// TIA Portal V20 export
FUNCTION_BLOCK "CallEquipment"   // FB43, LAD
TITLE = CallEquipment
// This block includes all general functions, checks and logik that is needed in the entire unit. E.g. general releases and system wide functionalities like air, pressure and power handling as well as general reaction to events.
// stored: IsIECCheckEnabled true, MemoryReserve 100, Namespace Unit1.Em5, SetENOAutomatically true
   VAR_INPUT
      ZoneOperationEnable { ExternalWritable := 'False'} : "LWONIK_typeSafetyZoneManualOperation";
   END_VAR
   VAR_IN_OUT
      unitStatus : "LAF_typeUnitStatus";   // Current unit status o be used in this EM
      emFeedback : "LUC_typeEmFeedback";   // Feedback of the EM to the Unit
      unitAlarmDB : "LAF_typeAlarms";   // Summarized EM Alarms for the Unit
   END_VAR
   VAR
      InstSequenceTransferPnPLeft { ExternalWritable := 'False'} : "Unit1.Em5.Sequence_1_TransferPnPLeft";
      InstSequenceTransferPnPRight { ExternalWritable := 'False'} : "Unit1.Em5.Sequence_2_TransferPnPRight";
      InstSequenceGaugeRnR { ExternalWritable := 'False'} : "Unit1.Em5.Sequence_10_GaugeRnR";
      instTransferPnPLeftHomeJob1 { ExternalWritable := 'False'} : "LAF_SelectJob";
      instTransferPnPLeftSideTapeLoadJob2 { ExternalWritable := 'False'} : "LAF_SelectJob";
      instTransferPnPLeftHotPressLeftUnloadJob3 { ExternalWritable := 'False'} : "LAF_SelectJob";
      instTransferPnPLeftHotPressLeftLoadJob4 { ExternalWritable := 'False'} : "LAF_SelectJob";
      instTransferPnPLeftSideTapeLoadJob5 { ExternalWritable := 'False'} : "LAF_SelectJob";
      instTransferPnPLeftHotPressRightUnloadJob6 { ExternalWritable := 'False'} : "LAF_SelectJob";
      instTransferPnPLeftHotPressRightLoadJob7 { ExternalWritable := 'False'} : "LAF_SelectJob";
      instTransferPnPLeftHipotThicknessUnloadJob9 { ExternalWritable := 'False'} : "LAF_SelectJob";
      instTransferPnPRightHomeJob1 { ExternalWritable := 'False'} : "LAF_SelectJob";
      instTransferPnPRightHipotThicknessLoadJob2 { ExternalWritable := 'False'} : "LAF_SelectJob";
      instTransferPnPRightVisionUnloadJob3 { ExternalWritable := 'False'} : "LAF_SelectJob";
      instTransferPnPRightVisionLoadJob4 { ExternalWritable := 'False'} : "LAF_SelectJob";
      instTransferPnPRightLaserMarkUnloadJob5 { ExternalWritable := 'False'} : "LAF_SelectJob";
      instTransferPnPRightLaserMarkLoadJob6 { ExternalWritable := 'False'} : "LAF_SelectJob";
      instTransferPnPRightWeightCheckUnloadJob9 { ExternalWritable := 'False'} : "LAF_SelectJob";
      instGRnR_SideTapeLoadJob2_Left { ExternalWritable := 'False'} : "LAF_SelectJob";
      instGRnR_HipotThicknessUnloadJob3_Left { ExternalWritable := 'False'} : "LAF_SelectJob";
      instGRnR_HipotThicknessLoadJob4_Left { ExternalWritable := 'False'} : "LAF_SelectJob";
      instGRnR_HipotThicknessLoadJob5_Right { ExternalWritable := 'False'} : "LAF_SelectJob";
      instGRnR_VisionUnloadJob6_Right { ExternalWritable := 'False'} : "LAF_SelectJob";
      instGRnR_VisionLoadJob7_Right { ExternalWritable := 'False'} : "LAF_SelectJob";
      instGRnR_WeightCheckUnloadJob8_Right { ExternalWritable := 'False'} : "LAF_SelectJob";
      instGRnR_WeightCheckLoadJob9_Right { ExternalWritable := 'False'} : "LAF_SelectJob";
      instCmTransferPnPLeftSafetyPin { ExternalWritable := 'False'} : "LBC_DigitalSignalCn";
      instCmTransferPnPLeftJRDetect { ExternalWritable := 'False'} : "LBC_DigitalSignalCn";
      instCmTransferPnPRightSafetyPin { ExternalWritable := 'False'} : "LBC_DigitalSignalCn";
      instCmTransferPnPRightJRDetect { ExternalWritable := 'False'} : "LBC_DigitalSignalCn";
      instCmTransferPnPLeftAxisX { ExternalWritable := 'False'} : "LBC_Axis64Pos_TecPlcCn";
      instCmTransferPnPLeftAxisY { ExternalWritable := 'False'} : "LBC_Axis64Pos_TecPlcCn";
      instCmTransferPnPLeftAxisZ { ExternalWritable := 'False'} : "LBC_Axis64Pos_TecPlcCn";
      instCmTransferPnPRightAxisX { ExternalWritable := 'False'} : "LBC_Axis64Pos_TecPlcCn";
      instCmTransferPnPRightAxisY { ExternalWritable := 'False'} : "LBC_Axis64Pos_TecPlcCn";
      instCmTransferPnPRightAxisZ { ExternalWritable := 'False'} : "LBC_Axis64Pos_TecPlcCn";
      instCmTransferPnPLeftClampOpenClose { ExternalWritable := 'False'} : "LBC_TwoWayActuatorCn";
      instCmTransferPnPRightClampOpenClose { ExternalWritable := 'False'} : "LBC_TwoWayActuatorCn";
      instInterlockTransferPnPLeftAxisX { ExternalWritable := 'False'} : "LER_Axis64Pos_InterlockSummary";
      instInterlockTransferPnPLeftAxisY { ExternalWritable := 'False'} : "LER_Axis64Pos_InterlockSummary";
      instInterlockTransferPnPLeftAxisZ { ExternalWritable := 'False'} : "LER_Axis64Pos_InterlockSummary";
      instInterlockTransferPnPRightAxisX { ExternalWritable := 'False'} : "LER_Axis64Pos_InterlockSummary";
      instInterlockTransferPnPRightAxisY { ExternalWritable := 'False'} : "LER_Axis64Pos_InterlockSummary";
      instInterlockTransferPnPRightAxisZ { ExternalWritable := 'False'} : "LER_Axis64Pos_InterlockSummary";
      instLDrv701ControlTransferPnPLeftAxisZ { ExternalWritable := 'False'} : "LDrvSafe_SinaTlg701Control";   // Drive Telegram Function Library
      instLDrv701StatusTransferPnPLeftAxisZ { ExternalWritable := 'False'} : "LDrvSafe_SinaTlg701Status";   // Drive Telegram Function Library
      instLDrv701ControlTransferPnPRightAxisZ { ExternalWritable := 'False'} : "LDrvSafe_SinaTlg701Control";   // Drive Telegram Function Library
      instLDrv701StatusTransferPnPRightAxisZ { ExternalWritable := 'False'} : "LDrvSafe_SinaTlg701Status";   // Drive Telegram Function Library
      instManageAlarms { ExternalWritable := 'False'} : "LAF_ManageAlarms";
      instEventsPFE { ExternalWritable := 'False'} : "Unit1.Em5.EventsPFE";
      statUnitStatus { ExternalWritable := 'False'} : "LAF_typeUnitStatus";   // Unit Status that is used in this project
      statSlmStatus { ExternalWritable := 'False'} : Struct
         running : Bool;
         powerOff : Bool;
      END_STRUCT;
      statAllBrakeTest { ExternalWritable := 'False'} : "LER_typeBrakeTestUnitCommands";
      statFlipFlop { ExternalWritable := 'False'} : Array[0..99] of Bool;
      statPartData { ExternalWritable := 'False'} : "LER_typePartData";
      statDataDelete { ExternalWritable := 'False'} : "LER_typePartData";
      statRoutingOk { ExternalWritable := 'False'} : Array[0..99] of Bool;
      statRoutingNok { ExternalWritable := 'False'} : Array[0..99] of Bool;
      statTonTime { ExternalWritable := 'False'} : Array[0..999] of TON_TIME;
      statTofTime { ExternalWritable := 'False'} : Array[0..99] of TOF_TIME;
      statPulse { ExternalWritable := 'False'} : Array[0..999] of Bool;
      statTrPnP_GaugeRnR : Struct
         currentCount : Int;
         processCount : Int;
         Ongoing : Bool;
         Complete : Bool;
      END_STRUCT;
      statEnableManualCmds { ExternalWritable := 'False'} : Bool;
      "*** Interlock Axis ***" : Bool;
      TransferPnPLeftAxisX_Home { S7_SetPoint := 'True'} : "LER_Axis_Homing";
      TransferPnPLeftAxisY_Home { S7_SetPoint := 'True'} : "LER_Axis_Homing";
      TransferPnPLeftAxisZ_Home { S7_SetPoint := 'True'} : "LER_Axis_Homing";
      TransferPnPRightAxisX_Home { S7_SetPoint := 'True'} : "LER_Axis_Homing";
      TransferPnPRightAxisY_Home { S7_SetPoint := 'True'} : "LER_Axis_Homing";
      TransferPnPRightAxisZ_Home { S7_SetPoint := 'True'} : "LER_Axis_Homing";
      TransferPnPLeftAxisX_IntHome : Array[0..9] of Bool;
      TransferPnPLeftAxisY_IntHome : Array[0..9] of Bool;
      TransferPnPLeftAxisZ_IntHome : Array[0..9] of Bool;
      TransferPnPRightAxisX_IntHome : Array[0..9] of Bool;
      TransferPnPRightAxisY_IntHome : Array[0..9] of Bool;
      TransferPnPRightAxisZ_IntHome : Array[0..9] of Bool;
      TransferPnPLeftAxisX_Jog { S7_SetPoint := 'True'} : Array[0..2] of "LER_Axis_Jog";
      TransferPnPLeftAxisY_Jog { S7_SetPoint := 'True'} : Array[0..2] of "LER_Axis_Jog";
      TransferPnPLeftAxisZ_Jog { S7_SetPoint := 'True'} : Array[0..2] of "LER_Axis_Jog";
      TransferPnPRightAxisX_Jog { S7_SetPoint := 'True'} : Array[0..2] of "LER_Axis_Jog";
      TransferPnPRightAxisY_Jog { S7_SetPoint := 'True'} : Array[0..2] of "LER_Axis_Jog";
      TransferPnPRightAxisZ_Jog { S7_SetPoint := 'True'} : Array[0..2] of "LER_Axis_Jog";
      TransferPnPLeftAxisX_interlock { S7_SetPoint := 'True'} : Array[0..10] of "LER_Axis_Absolute";
      TransferPnPLeftAxisY_interlock { S7_SetPoint := 'True'} : Array[0..10] of "LER_Axis_Absolute";
      TransferPnPLeftAxisZ_interlock { S7_SetPoint := 'True'} : Array[0..10] of "LER_Axis_Absolute";
      TransferPnPRightAxisX_interlock { S7_SetPoint := 'True'} : Array[0..10] of "LER_Axis_Absolute";
      TransferPnPRightAxisY_interlock { S7_SetPoint := 'True'} : Array[0..10] of "LER_Axis_Absolute";
      TransferPnPRightAxisZ_interlock { S7_SetPoint := 'True'} : Array[0..10] of "LER_Axis_Absolute";
      TransferPnPLeftAxisX_IntPos : Array[0..9] of Struct
         "Int" : Array[1..10] of Bool;
      END_STRUCT;
      TransferPnPLeftAxisY_IntPos : Array[0..9] of Struct
         "Int" : Array[1..10] of Bool;
      END_STRUCT;
      TransferPnPLeftAxisZ_IntPos : Array[0..9] of Struct
         "Int" : Array[1..10] of Bool;
      END_STRUCT;
      TransferPnPRightAxisX_IntPos : Array[0..9] of Struct
         "Int" : Array[1..10] of Bool;
      END_STRUCT;
      TransferPnPRightAxisY_IntPos : Array[0..9] of Struct
         "Int" : Array[1..10] of Bool;
      END_STRUCT;
      TransferPnPRightAxisZ_IntPos : Array[0..9] of Struct
         "Int" : Array[1..10] of Bool;
      END_STRUCT;
      "*** Interlock TwoWay ***" { S7_SetPoint := 'True'} : "LER_Axis_Homing";
      instCmTransferPnPLeftClampOpenCloseInterlock { S7_SetPoint := 'True'} : Array[0..2] of "LER_Actuator";
      instCmTransferPnPRightClampOpenCloseInterlock { S7_SetPoint := 'True'} : Array[0..2] of "LER_Actuator";
      TransferPnPLeftClampOpenClose_Inpos : Array[0..2] of Struct
         "Int" : Array[1..10] of Bool;
      END_STRUCT;
      TransferPnPRightClampOpenClose_Inpos : Array[0..2] of Struct
         "Int" : Array[1..10] of Bool;
      END_STRUCT;
      citi_Ptrig : Array[0..20] of Bool;
      citiTon : Array[0..20] of TON_TIME;
      citi : Time;
      citiTest : Array[0..20] of Bool;
   END_VAR
   VAR_TEMP
      tempScInProduction : Bool;   // Mode Production and StateComplete
      tempScNoProduction : Bool;   // Mode Manual and StateComplete
      tempPnPLeftPart_No_Detect : Bool;
      tempPnPRightPart_No_Detect : Bool;
      tempPnPLeftPart_Detect : Bool;
      tempPnPRightPart_Detect : Bool;
      tempGuageRnR_1CycleDone : Bool;
      tempSpecialFunctionCheckbit : Bool;
      tempInterlockCond : Bool;
      tempPickCond : Bool;
      tempPlaceCond : Bool;
   END_VAR
   VAR CONSTANT
      delayTime : Time := T#3s;
      TRUE : Bool := TRUE;
      FALSE : Bool := FALSE;
      NO_JOB : DInt;
      MIN_POSITION_NUMBER : SInt;
      INIT_POSITION_NUMBER : SInt := -1;
      Stacker1 : Char := 'A';
      Stacker2 : Char := 'B';
   END_VAR
   VAR_TEMP   // added for the SCL form of the ladder/FBD networks
      _w1 : Bool;
      _w2 : Bool;
      _w3 : Bool;
      _w4 : Bool;
      _w5 : Bool;
      _w6 : Bool;
      _w7 : Bool;
      _w8 : Bool;
      _w9 : Bool;
      _w10 : Bool;
      _w11 : Bool;
      _w12 : Bool;
      _w13 : Bool;
      _w14 : Bool;
      _w15 : Bool;
      _w16 : Bool;
   END_VAR
BEGIN

REGION Network 1: BLOCK INFO HEADER
   // (company) / (C) Copyright (year)
   // ---------------------------------------------------------------------------------
   // Title:                             (Title of this block)
   // Comment/Function: (that is implemented in the block)
   // Library/Family:           (that the source is dedicated to)
   // Author:                        (department / person in charge / contact)
   // Target System:          (test system with FW version)
   // Engineering:              TIA Portal (SW version)
   // Restrictions:               (OB types, etc.)
   // Requirements:           (hardware, technological package, etc.)
   // ---------------------------------------------------------------------------------
   // Change log table:
   // Version          | Date             | Signature      | Expert in charge  | Changes applied ------------------------|----------------------|-------------------------|--------------------------------|-----------------------
   // 001.000.000 | yyyy-mm-dd | 0x00000000 | (name of expert) | First released version
END_REGION

REGION Network 2: DESCRIPTION
   // This is a template block provided by the Automation Framework. It can be used to create an own project.
   // The Block Info Header is prepared to put in your own data.
   // Description of the block could be added here and the docu created by Code2Docu.
END_REGION

REGION Network 3: Simulation
   // If simulation is active on a global level, inherit this status and set simulation active in this unit also. Information is written to DB ControlNodes, from where it is distributed to the equipmemt modules.
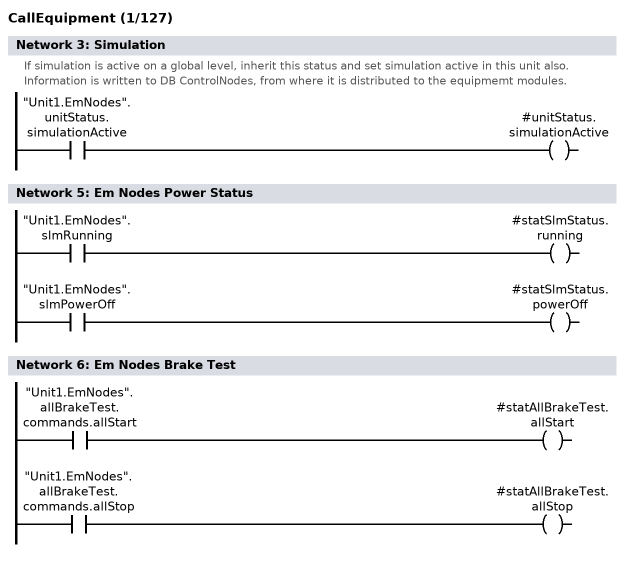
   RUNG wire#powerrail
      Contact( "Unit1.EmNodes".unitStatus.simulationActive )
      Coil( #unitStatus.simulationActive )
   END_RUNG
   // the same network as SCL:
   #unitStatus.simulationActive := "Unit1.EmNodes".unitStatus.simulationActive;
END_REGION

REGION Network 4: ******************** Unit Input ********************
END_REGION

REGION Network 5: Em Nodes Power Status
   RUNG wire#powerrail
      Contact( "Unit1.EmNodes".slmRunning )
      Coil( #statSlmStatus.running )
   END_RUNG
   RUNG wire#powerrail
      Contact( "Unit1.EmNodes".slmPowerOff )
      Coil( #statSlmStatus.powerOff )
   END_RUNG
   // the same network as SCL:
   #statSlmStatus.running := "Unit1.EmNodes".slmRunning;
   #statSlmStatus.powerOff := "Unit1.EmNodes".slmPowerOff;
END_REGION

REGION Network 6: Em Nodes Brake Test
   RUNG wire#powerrail
      Contact( "Unit1.EmNodes".allBrakeTest.commands.allStart )
      Coil( #statAllBrakeTest.allStart )
   END_RUNG
   RUNG wire#powerrail
      Contact( "Unit1.EmNodes".allBrakeTest.commands.allStop )
      Coil( #statAllBrakeTest.allStop )
   END_RUNG
   // the same network as SCL:
   #statAllBrakeTest.allStart := "Unit1.EmNodes".allBrakeTest.commands.allStart;
   #statAllBrakeTest.allStop := "Unit1.EmNodes".allBrakeTest.commands.allStop;
END_REGION

REGION Network 7: Em Data
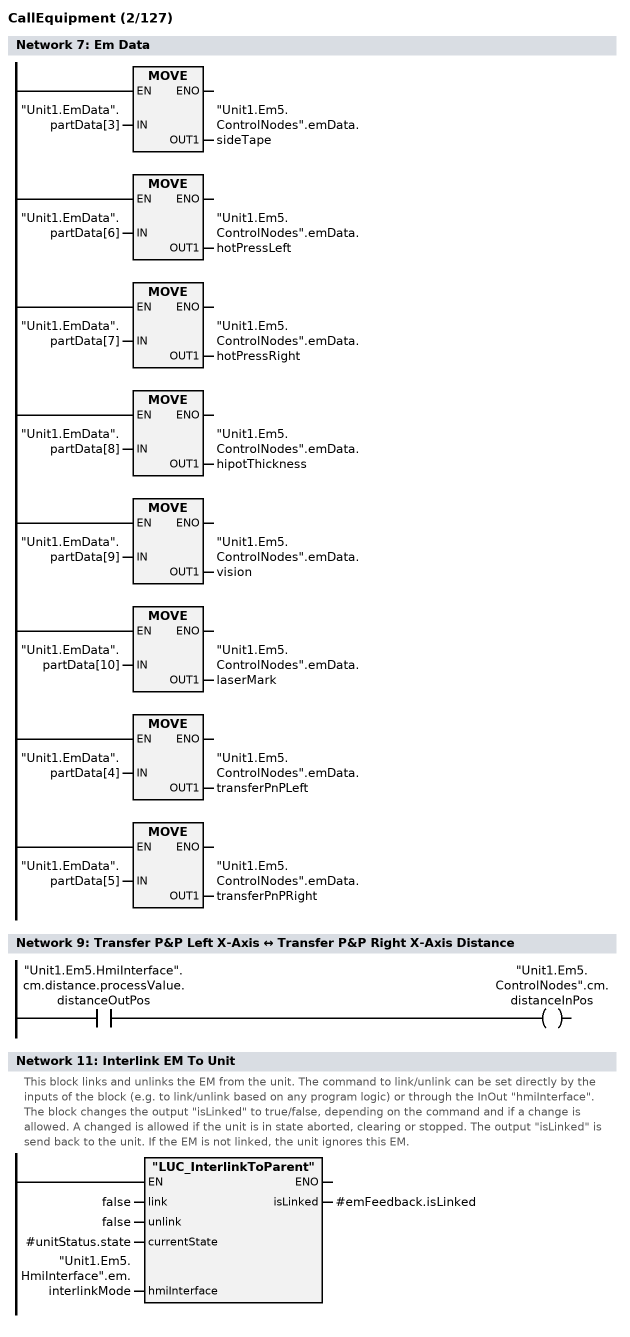
   RUNG wire#powerrail
      Move(in := "Unit1.EmData".partData[3], out1 => "Unit1.Em5.ControlNodes".emData.sideTape)
   END_RUNG
   RUNG wire#powerrail
      Move(in := "Unit1.EmData".partData[6], out1 => "Unit1.Em5.ControlNodes".emData.hotPressLeft)
   END_RUNG
   RUNG wire#powerrail
      Move(in := "Unit1.EmData".partData[7], out1 => "Unit1.Em5.ControlNodes".emData.hotPressRight)
   END_RUNG
   RUNG wire#powerrail
      Move(in := "Unit1.EmData".partData[8], out1 => "Unit1.Em5.ControlNodes".emData.hipotThickness)
   END_RUNG
   RUNG wire#powerrail
      Move(in := "Unit1.EmData".partData[9], out1 => "Unit1.Em5.ControlNodes".emData.vision)
   END_RUNG
   RUNG wire#powerrail
      Move(in := "Unit1.EmData".partData[10], out1 => "Unit1.Em5.ControlNodes".emData.laserMark)
   END_RUNG
   RUNG wire#powerrail
      Move(in := "Unit1.EmData".partData[4], out1 => "Unit1.Em5.ControlNodes".emData.transferPnPLeft)
   END_RUNG
   RUNG wire#powerrail
      Move(in := "Unit1.EmData".partData[5], out1 => "Unit1.Em5.ControlNodes".emData.transferPnPRight)
   END_RUNG
   // the same network as SCL:
   "Unit1.Em5.ControlNodes".emData.sideTape := "Unit1.EmData".partData[3];
   "Unit1.Em5.ControlNodes".emData.hotPressLeft := "Unit1.EmData".partData[6];
   "Unit1.Em5.ControlNodes".emData.hotPressRight := "Unit1.EmData".partData[7];
   "Unit1.Em5.ControlNodes".emData.hipotThickness := "Unit1.EmData".partData[8];
   "Unit1.Em5.ControlNodes".emData.vision := "Unit1.EmData".partData[9];
   "Unit1.Em5.ControlNodes".emData.laserMark := "Unit1.EmData".partData[10];
   "Unit1.Em5.ControlNodes".emData.transferPnPLeft := "Unit1.EmData".partData[4];
   "Unit1.Em5.ControlNodes".emData.transferPnPRight := "Unit1.EmData".partData[5];
END_REGION

REGION Network 8: ******************** HmiInterface → ControlNode ********************
END_REGION

REGION Network 9: Transfer P&P Left X-Axis ↔ Transfer P&P Right X-Axis Distance
   RUNG wire#powerrail
      Contact( "Unit1.Em5.HmiInterface".cm.distance.processValue.distanceOutPos )
      Coil( "Unit1.Em5.ControlNodes".cm.distanceInPos )
   END_RUNG
   // the same network as SCL:
   "Unit1.Em5.ControlNodes".cm.distanceInPos := "Unit1.Em5.HmiInterface".cm.distance.processValue.distanceOutPos;
END_REGION

REGION Network 10: ******************** Equipment Control ********************
END_REGION

REGION Network 11: Interlink EM To Unit
   // This block links and unlinks the EM from the unit. The command to link/unlink can be set directly by the inputs of the block (e.g. to link/unlink based on any program logic) or through the InOut "hmiInterface". The block changes the output "isLinked" to true/false, depending on the command and if a change is allowed. A changed is allowed if the unit is in state aborted, clearing or stopped. The output "isLinked" is send back to the unit. If the EM is not linked, the unit ignores this EM.
   RUNG wire#powerrail
      "LUC_InterlinkToParent"(link := false, unlink := false, currentState := #unitStatus.state, hmiInterface := "Unit1.Em5.HmiInterface".em.interlinkMode, isLinked => #emFeedback.isLinked)
   END_RUNG
   // the same network as SCL:
   "LUC_InterlinkToParent"(link := false,
                           unlink := false,
                           currentState := #unitStatus.state,
                           hmiInterface := "Unit1.Em5.HmiInterface".em.interlinkMode,
                           isLinked => #emFeedback.isLinked);
END_REGION

REGION Network 12: Control EM
   // When linked, unitStatus is fully applied to unitStatusUsed.
   // When not linked, only acknowledge and safetyReleased from the unitStatus are applied. A direct EM control by hmiInterface or localInterface is possible.
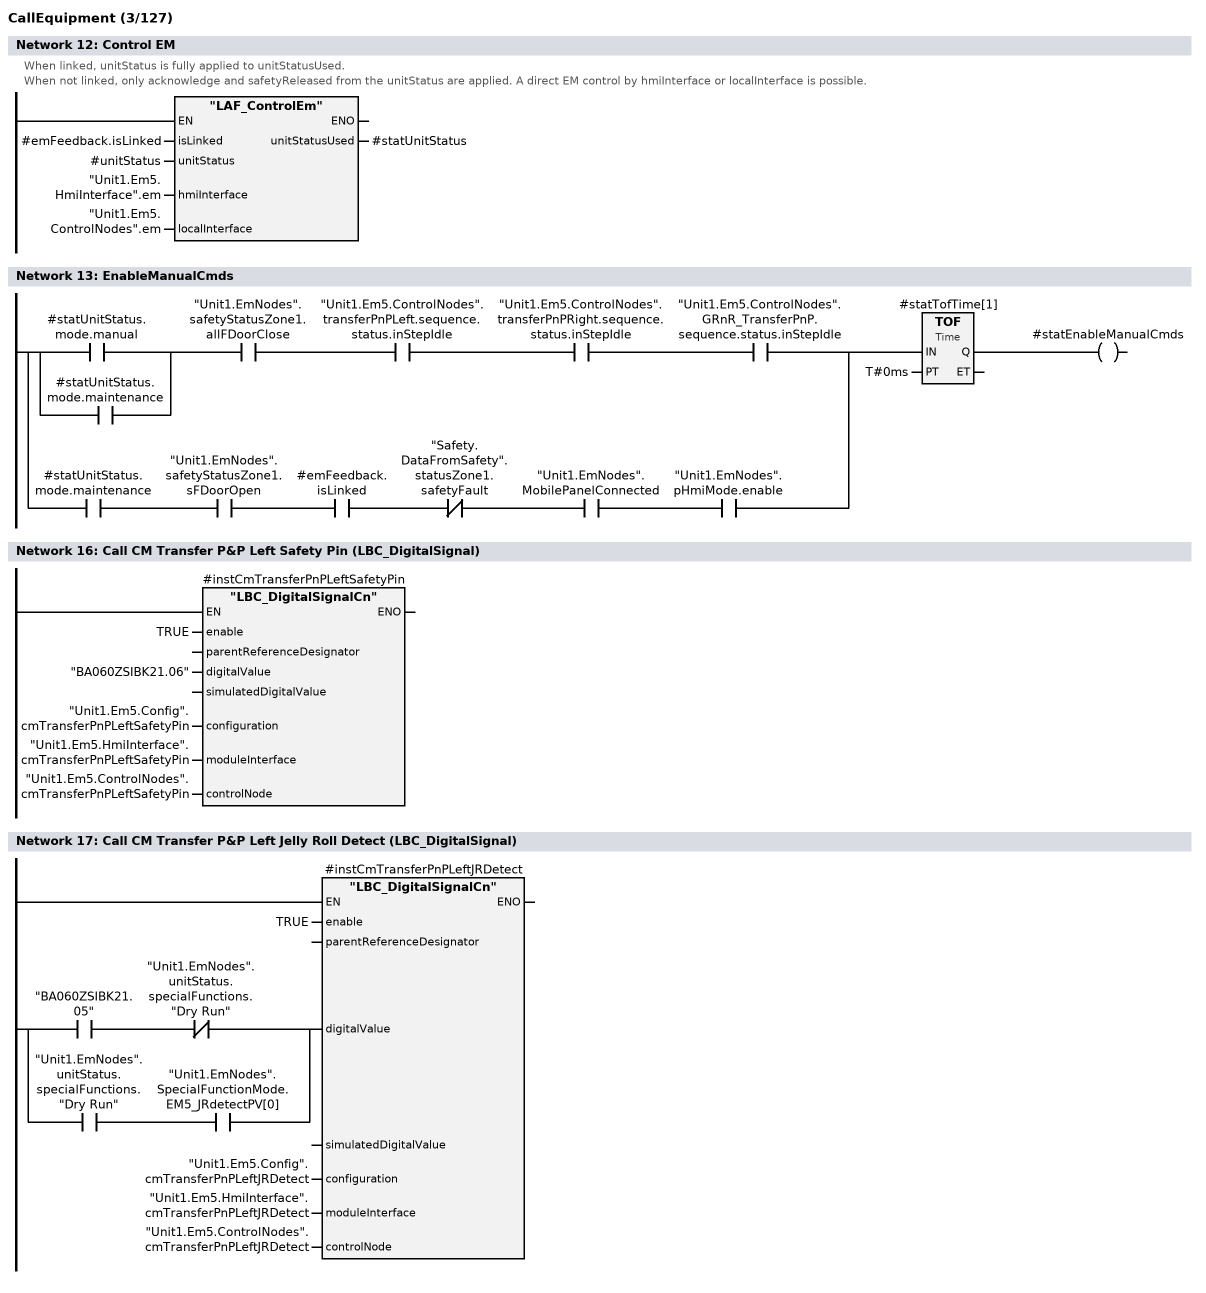
   RUNG wire#powerrail
      "LAF_ControlEm"(isLinked := #emFeedback.isLinked, unitStatus := #unitStatus, hmiInterface := "Unit1.Em5.HmiInterface".em, localInterface := "Unit1.Em5.ControlNodes".em, unitStatusUsed => #statUnitStatus)
   END_RUNG
   // the same network as SCL:
   "LAF_ControlEm"(isLinked := #emFeedback.isLinked,
                   unitStatus := #unitStatus,
                   hmiInterface := "Unit1.Em5.HmiInterface".em,
                   localInterface := "Unit1.Em5.ControlNodes".em,
                   unitStatusUsed => #statUnitStatus);
END_REGION

REGION Network 13: EnableManualCmds
   RUNG wire#powerrail
      Contact( #statUnitStatus.mode.manual )
      wire#w1
      Contact( "Unit1.EmNodes".safetyStatusZone1.allFDoorClose )
      Contact( "Unit1.Em5.ControlNodes".transferPnPLeft.sequence.status.inStepIdle )
      Contact( "Unit1.Em5.ControlNodes".transferPnPRight.sequence.status.inStepIdle )
      Contact( "Unit1.Em5.ControlNodes".GRnR_TransferPnP.sequence.status.inStepIdle )
      wire#w2
      { S7_Templates := "time_type := Time" } #statTofTime[1].TOF(pt := T#0ms, et =>)
      Coil( #statEnableManualCmds )
   END_RUNG
   RUNG wire#powerrail
      Contact( #statUnitStatus.mode.maintenance )
   END_RUNG wire#w1
   RUNG wire#powerrail
      Contact( #statUnitStatus.mode.maintenance )
      Contact( "Unit1.EmNodes".safetyStatusZone1.sFDoorOpen )
      Contact( #emFeedback.isLinked )
      I_Contact( "Safety.DataFromSafety".statusZone1.safetyFault )
      Contact( "Unit1.EmNodes".MobilePanelConnected )
      Contact( "Unit1.EmNodes".pHmiMode.enable )
   END_RUNG wire#w2
   // the same network as SCL:
   #statTofTime[1].TOF(IN := ((#statUnitStatus.mode.manual OR #statUnitStatus.mode.maintenance) AND "Unit1.EmNodes".safetyStatusZone1.allFDoorClose AND "Unit1.Em5.ControlNodes".transferPnPLeft.sequence.status.inStepIdle AND "Unit1.Em5.ControlNodes".transferPnPRight.sequence.status.inStepIdle AND "Unit1.Em5.ControlNodes".GRnR_TransferPnP.sequence.status.inStepIdle) OR (#statUnitStatus.mode.maintenance AND "Unit1.EmNodes".safetyStatusZone1.sFDoorOpen AND #emFeedback.isLinked AND NOT "Safety.DataFromSafety".statusZone1.safetyFault AND "Unit1.EmNodes".MobilePanelConnected AND "Unit1.EmNodes".pHmiMode.enable),
                       PT := T#0ms);
   #statEnableManualCmds := #statTofTime[1].Q;
END_REGION

REGION Network 15: ******************** Control Modules (Sensors) ********************
   // Call control modules that are sensors before the em logic (jobs and sequence), so that the latest value is used in the logic.
END_REGION

REGION Network 16: Call CM Transfer P&P Left Safety Pin (LBC_DigitalSignal)
   RUNG wire#powerrail
      #instCmTransferPnPLeftSafetyPin(enable := TRUE, parentReferenceDesignator :=, digitalValue := "BA060ZSIBK21.06", simulatedDigitalValue :=, configuration := "Unit1.Em5.Config".cmTransferPnPLeftSafetyPin, moduleInterface := "Unit1.Em5.HmiInterface".cmTransferPnPLeftSafetyPin, controlNode := "Unit1.Em5.ControlNodes".cmTransferPnPLeftSafetyPin)
   END_RUNG
   // the same network as SCL:
   #instCmTransferPnPLeftSafetyPin(enable := TRUE,   // "LBC_DigitalSignalCn"
                           digitalValue := "BA060ZSIBK21.06",
                           configuration := "Unit1.Em5.Config".cmTransferPnPLeftSafetyPin,
                           moduleInterface := "Unit1.Em5.HmiInterface".cmTransferPnPLeftSafetyPin,
                           controlNode := "Unit1.Em5.ControlNodes".cmTransferPnPLeftSafetyPin);
END_REGION

REGION Network 17: Call CM Transfer P&P Left Jelly Roll Detect (LBC_DigitalSignal)
   RUNG wire#powerrail
      #instCmTransferPnPLeftJRDetect(digitalValue := wire#w1, enable := TRUE, parentReferenceDesignator :=, simulatedDigitalValue :=, configuration := "Unit1.Em5.Config".cmTransferPnPLeftJRDetect, moduleInterface := "Unit1.Em5.HmiInterface".cmTransferPnPLeftJRDetect, controlNode := "Unit1.Em5.ControlNodes".cmTransferPnPLeftJRDetect)
   END_RUNG
   RUNG wire#powerrail
      Contact( "BA060ZSIBK21.05" )
      I_Contact( "Unit1.EmNodes".unitStatus.specialFunctions."Dry Run" )
   END_RUNG wire#w1
   RUNG wire#powerrail
      Contact( "Unit1.EmNodes".unitStatus.specialFunctions."Dry Run" )
      Contact( "Unit1.EmNodes".SpecialFunctionMode.EM5_JRdetectPV[0] )
   END_RUNG wire#w1
   // the same network as SCL:
   #instCmTransferPnPLeftJRDetect(enable := TRUE,   // "LBC_DigitalSignalCn"
                           digitalValue := ("BA060ZSIBK21.05" AND NOT "Unit1.EmNodes".unitStatus.specialFunctions."Dry Run") OR ("Unit1.EmNodes".unitStatus.specialFunctions."Dry Run" AND "Unit1.EmNodes".SpecialFunctionMode.EM5_JRdetectPV[0]),
                           configuration := "Unit1.Em5.Config".cmTransferPnPLeftJRDetect,
                           moduleInterface := "Unit1.Em5.HmiInterface".cmTransferPnPLeftJRDetect,
                           controlNode := "Unit1.Em5.ControlNodes".cmTransferPnPLeftJRDetect);
END_REGION

REGION Network 18: Call CM Transfer P&P Right Safety Pin (LBC_DigitalSignal)
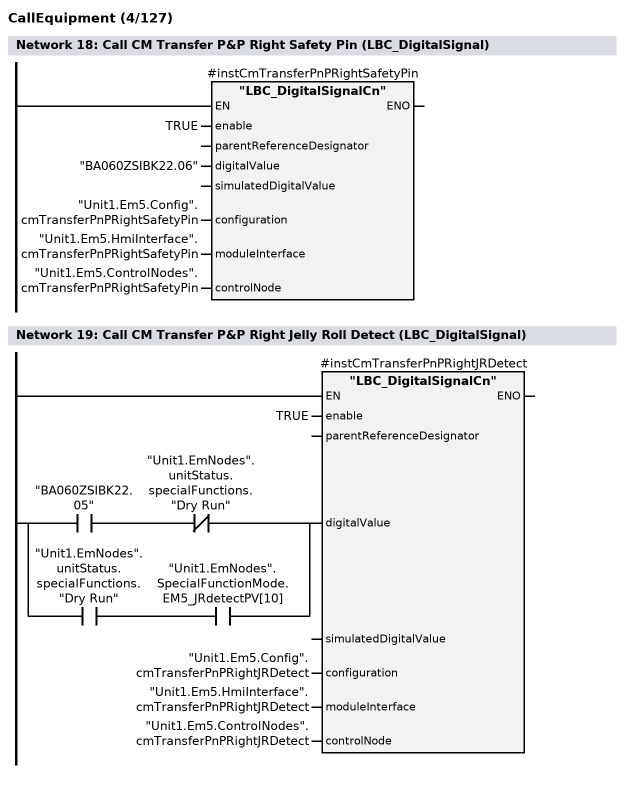
   RUNG wire#powerrail
      #instCmTransferPnPRightSafetyPin(enable := TRUE, parentReferenceDesignator :=, digitalValue := "BA060ZSIBK22.06", simulatedDigitalValue :=, configuration := "Unit1.Em5.Config".cmTransferPnPRightSafetyPin, moduleInterface := "Unit1.Em5.HmiInterface".cmTransferPnPRightSafetyPin, controlNode := "Unit1.Em5.ControlNodes".cmTransferPnPRightSafetyPin)
   END_RUNG
   // the same network as SCL:
   #instCmTransferPnPRightSafetyPin(enable := TRUE,   // "LBC_DigitalSignalCn"
                           digitalValue := "BA060ZSIBK22.06",
                           configuration := "Unit1.Em5.Config".cmTransferPnPRightSafetyPin,
                           moduleInterface := "Unit1.Em5.HmiInterface".cmTransferPnPRightSafetyPin,
                           controlNode := "Unit1.Em5.ControlNodes".cmTransferPnPRightSafetyPin);
END_REGION

REGION Network 19: Call CM Transfer P&P Right Jelly Roll Detect (LBC_DigitalSignal)
   RUNG wire#powerrail
      #instCmTransferPnPRightJRDetect(digitalValue := wire#w1, enable := TRUE, parentReferenceDesignator :=, simulatedDigitalValue :=, configuration := "Unit1.Em5.Config".cmTransferPnPRightJRDetect, moduleInterface := "Unit1.Em5.HmiInterface".cmTransferPnPRightJRDetect, controlNode := "Unit1.Em5.ControlNodes".cmTransferPnPRightJRDetect)
   END_RUNG
   RUNG wire#powerrail
      Contact( "BA060ZSIBK22.05" )
      I_Contact( "Unit1.EmNodes".unitStatus.specialFunctions."Dry Run" )
   END_RUNG wire#w1
   RUNG wire#powerrail
      Contact( "Unit1.EmNodes".unitStatus.specialFunctions."Dry Run" )
      Contact( "Unit1.EmNodes".SpecialFunctionMode.EM5_JRdetectPV[10] )
   END_RUNG wire#w1
   // the same network as SCL:
   #instCmTransferPnPRightJRDetect(enable := TRUE,   // "LBC_DigitalSignalCn"
                           digitalValue := ("BA060ZSIBK22.05" AND NOT "Unit1.EmNodes".unitStatus.specialFunctions."Dry Run") OR ("Unit1.EmNodes".unitStatus.specialFunctions."Dry Run" AND "Unit1.EmNodes".SpecialFunctionMode.EM5_JRdetectPV[10]),
                           configuration := "Unit1.Em5.Config".cmTransferPnPRightJRDetect,
                           moduleInterface := "Unit1.Em5.HmiInterface".cmTransferPnPRightJRDetect,
                           controlNode := "Unit1.Em5.ControlNodes".cmTransferPnPRightJRDetect);
END_REGION

REGION Network 21: ******************** Equipment seuqnece logic ********************
END_REGION

REGION Network 22: Map Unit Status To Sequence Status
   // This block maps the unit status to the seuqnce status. Thus, it controls the sequence depending on the unit status. E.g. it sets the sequence to automatic when the unit state is in productions. This blocks work perfectly with the sequences provided in the AF. 
   // This typed block (MapUnitStatusToSequence) could be adjusted to specific application requirements or if other, user-defined sequences are used.
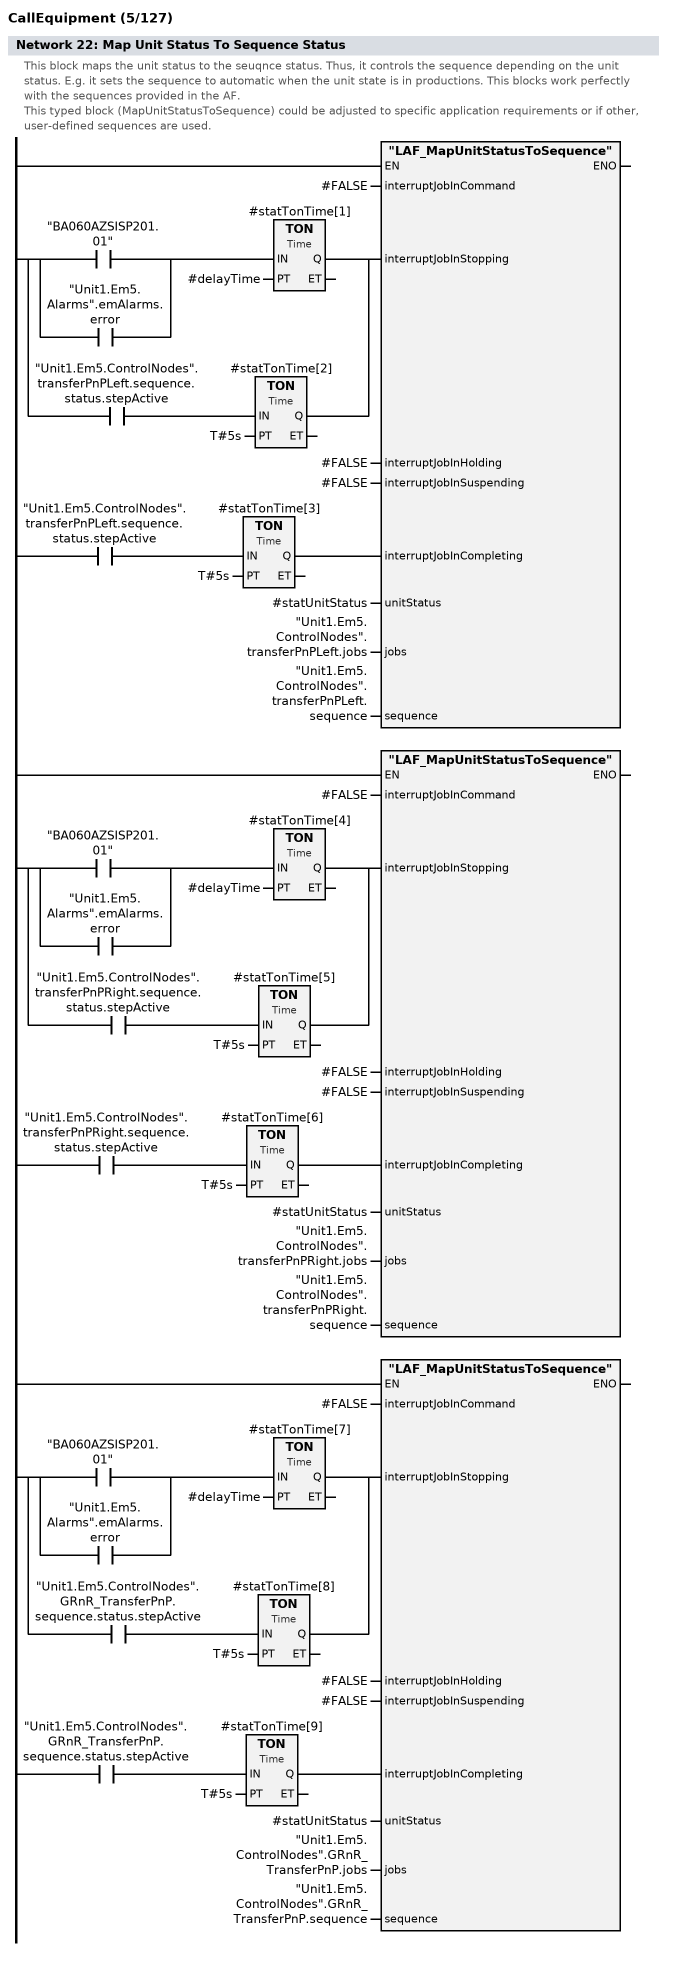
   RUNG wire#powerrail
      "LAF_MapUnitStatusToSequence"(interruptJobInStopping := wire#w2, interruptJobInCompleting := wire#w3, interruptJobInCommand := #FALSE, interruptJobInHolding := #FALSE, interruptJobInSuspending := #FALSE, unitStatus := #statUnitStatus, jobs := "Unit1.Em5.ControlNodes".transferPnPLeft.jobs, sequence := "Unit1.Em5.ControlNodes".transferPnPLeft.sequence)
   END_RUNG
   RUNG wire#powerrail
      Contact( "BA060AZSISP201.01" )
      wire#w1
      { S7_Templates := "time_type := Time" } #statTonTime[1].TON(pt := #delayTime, et =>)
   END_RUNG wire#w2
   RUNG wire#powerrail
      Contact( "Unit1.Em5.Alarms".emAlarms.error )
   END_RUNG wire#w1
   RUNG wire#powerrail
      Contact( "Unit1.Em5.ControlNodes".transferPnPLeft.sequence.status.stepActive )
      { S7_Templates := "time_type := Time" } #statTonTime[2].TON(pt := T#5s, et =>)
   END_RUNG wire#w2
   RUNG wire#powerrail
      Contact( "Unit1.Em5.ControlNodes".transferPnPLeft.sequence.status.stepActive )
      { S7_Templates := "time_type := Time" } #statTonTime[3].TON(pt := T#5s, et =>)
   END_RUNG wire#w3
   RUNG wire#powerrail
      "LAF_MapUnitStatusToSequence"(interruptJobInStopping := wire#w5, interruptJobInCompleting := wire#w6, interruptJobInCommand := #FALSE, interruptJobInHolding := #FALSE, interruptJobInSuspending := #FALSE, unitStatus := #statUnitStatus, jobs := "Unit1.Em5.ControlNodes".transferPnPRight.jobs, sequence := "Unit1.Em5.ControlNodes".transferPnPRight.sequence)
   END_RUNG
   RUNG wire#powerrail
      Contact( "BA060AZSISP201.01" )
      wire#w4
      { S7_Templates := "time_type := Time" } #statTonTime[4].TON(pt := #delayTime, et =>)
   END_RUNG wire#w5
   RUNG wire#powerrail
      Contact( "Unit1.Em5.Alarms".emAlarms.error )
   END_RUNG wire#w4
   RUNG wire#powerrail
      Contact( "Unit1.Em5.ControlNodes".transferPnPRight.sequence.status.stepActive )
      { S7_Templates := "time_type := Time" } #statTonTime[5].TON(pt := T#5s, et =>)
   END_RUNG wire#w5
   RUNG wire#powerrail
      Contact( "Unit1.Em5.ControlNodes".transferPnPRight.sequence.status.stepActive )
      { S7_Templates := "time_type := Time" } #statTonTime[6].TON(pt := T#5s, et =>)
   END_RUNG wire#w6
   RUNG wire#powerrail
      "LAF_MapUnitStatusToSequence"(interruptJobInStopping := wire#w8, interruptJobInCompleting := wire#w9, interruptJobInCommand := #FALSE, interruptJobInHolding := #FALSE, interruptJobInSuspending := #FALSE, unitStatus := #statUnitStatus, jobs := "Unit1.Em5.ControlNodes".GRnR_TransferPnP.jobs, sequence := "Unit1.Em5.ControlNodes".GRnR_TransferPnP.sequence)
   END_RUNG
   RUNG wire#powerrail
      Contact( "BA060AZSISP201.01" )
      wire#w7
      { S7_Templates := "time_type := Time" } #statTonTime[7].TON(pt := #delayTime, et =>)
   END_RUNG wire#w8
   RUNG wire#powerrail
      Contact( "Unit1.Em5.Alarms".emAlarms.error )
   END_RUNG wire#w7
   RUNG wire#powerrail
      Contact( "Unit1.Em5.ControlNodes".GRnR_TransferPnP.sequence.status.stepActive )
      { S7_Templates := "time_type := Time" } #statTonTime[8].TON(pt := T#5s, et =>)
   END_RUNG wire#w8
   RUNG wire#powerrail
      Contact( "Unit1.Em5.ControlNodes".GRnR_TransferPnP.sequence.status.stepActive )
      { S7_Templates := "time_type := Time" } #statTonTime[9].TON(pt := T#5s, et =>)
   END_RUNG wire#w9
   // the same network as SCL:
   #statTonTime[1].TON(IN := "BA060AZSISP201.01" OR "Unit1.Em5.Alarms".emAlarms.error, PT := #delayTime);
   #_w1 := #statTonTime[1].Q;
   #statTonTime[2].TON(IN := "Unit1.Em5.ControlNodes".transferPnPLeft.sequence.status.stepActive, PT := T#5s);
   #_w2 := #_w1 OR #statTonTime[2].Q;
   #statTonTime[3].TON(IN := "Unit1.Em5.ControlNodes".transferPnPLeft.sequence.status.stepActive, PT := T#5s);
   "LAF_MapUnitStatusToSequence"(interruptJobInCommand := #FALSE,
                           interruptJobInStopping := #_w2,
                           interruptJobInHolding := #FALSE,
                           interruptJobInSuspending := #FALSE,
                           interruptJobInCompleting := #statTonTime[3].Q,
                           unitStatus := #statUnitStatus,
                           jobs := "Unit1.Em5.ControlNodes".transferPnPLeft.jobs,
                           sequence := "Unit1.Em5.ControlNodes".transferPnPLeft.sequence);
   #statTonTime[4].TON(IN := "BA060AZSISP201.01" OR "Unit1.Em5.Alarms".emAlarms.error, PT := #delayTime);
   #_w3 := #statTonTime[4].Q;
   #statTonTime[5].TON(IN := "Unit1.Em5.ControlNodes".transferPnPRight.sequence.status.stepActive, PT := T#5s);
   #_w4 := #_w3 OR #statTonTime[5].Q;
   #statTonTime[6].TON(IN := "Unit1.Em5.ControlNodes".transferPnPRight.sequence.status.stepActive, PT := T#5s);
   "LAF_MapUnitStatusToSequence"(interruptJobInCommand := #FALSE,
                           interruptJobInStopping := #_w4,
                           interruptJobInHolding := #FALSE,
                           interruptJobInSuspending := #FALSE,
                           interruptJobInCompleting := #statTonTime[6].Q,
                           unitStatus := #statUnitStatus,
                           jobs := "Unit1.Em5.ControlNodes".transferPnPRight.jobs,
                           sequence := "Unit1.Em5.ControlNodes".transferPnPRight.sequence);
   #statTonTime[7].TON(IN := "BA060AZSISP201.01" OR "Unit1.Em5.Alarms".emAlarms.error, PT := #delayTime);
   #_w5 := #statTonTime[7].Q;
   #statTonTime[8].TON(IN := "Unit1.Em5.ControlNodes".GRnR_TransferPnP.sequence.status.stepActive, PT := T#5s);
   #_w6 := #_w5 OR #statTonTime[8].Q;
   #statTonTime[9].TON(IN := "Unit1.Em5.ControlNodes".GRnR_TransferPnP.sequence.status.stepActive, PT := T#5s);
   "LAF_MapUnitStatusToSequence"(interruptJobInCommand := #FALSE,
                           interruptJobInStopping := #_w6,
                           interruptJobInHolding := #FALSE,
                           interruptJobInSuspending := #FALSE,
                           interruptJobInCompleting := #statTonTime[9].Q,
                           unitStatus := #statUnitStatus,
                           jobs := "Unit1.Em5.ControlNodes".GRnR_TransferPnP.jobs,
                           sequence := "Unit1.Em5.ControlNodes".GRnR_TransferPnP.sequence);
END_REGION

REGION Network 23: Special Function check bit
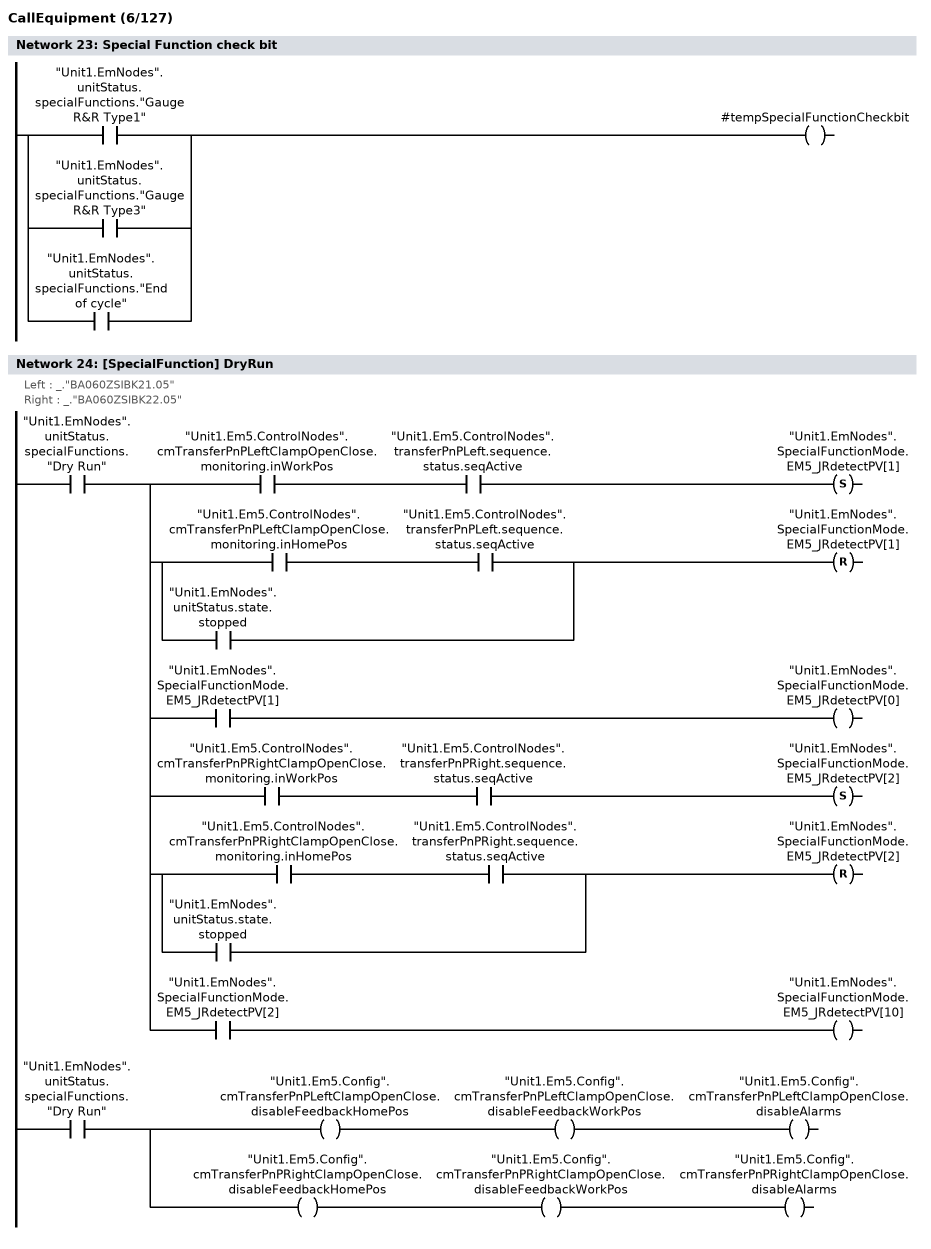
   RUNG wire#powerrail
      Contact( "Unit1.EmNodes".unitStatus.specialFunctions."Gauge R&R Type1" )
      wire#w1
      Coil( #tempSpecialFunctionCheckbit )
   END_RUNG
   RUNG wire#powerrail
      Contact( "Unit1.EmNodes".unitStatus.specialFunctions."Gauge R&R Type3" )
   END_RUNG wire#w1
   RUNG wire#powerrail
      Contact( "Unit1.EmNodes".unitStatus.specialFunctions."End of cycle" )
   END_RUNG wire#w1
   // the same network as SCL:
   #tempSpecialFunctionCheckbit := "Unit1.EmNodes".unitStatus.specialFunctions."Gauge R&R Type1" OR "Unit1.EmNodes".unitStatus.specialFunctions."Gauge R&R Type3" OR "Unit1.EmNodes".unitStatus.specialFunctions."End of cycle";
END_REGION

REGION Network 24: [SpecialFunction] DryRun
   // Left : _."BA060ZSIBK21.05"
   // Right : _."BA060ZSIBK22.05"
   RUNG wire#powerrail
      Contact( "Unit1.EmNodes".unitStatus.specialFunctions."Dry Run" )
      wire#w1
      Contact( "Unit1.Em5.ControlNodes".cmTransferPnPLeftClampOpenClose.monitoring.inWorkPos )
      Contact( "Unit1.Em5.ControlNodes".transferPnPLeft.sequence.status.seqActive )
      S_Coil( "Unit1.EmNodes".SpecialFunctionMode.EM5_JRdetectPV[1] )
   END_RUNG
   RUNG wire#w1
      Contact( "Unit1.Em5.ControlNodes".cmTransferPnPLeftClampOpenClose.monitoring.inHomePos )
      Contact( "Unit1.Em5.ControlNodes".transferPnPLeft.sequence.status.seqActive )
      wire#w2
      R_Coil( "Unit1.EmNodes".SpecialFunctionMode.EM5_JRdetectPV[1] )
   END_RUNG
   RUNG wire#w1
      Contact( "Unit1.EmNodes".unitStatus.state.stopped )
   END_RUNG wire#w2
   RUNG wire#w1
      Contact( "Unit1.EmNodes".SpecialFunctionMode.EM5_JRdetectPV[1] )
      Coil( "Unit1.EmNodes".SpecialFunctionMode.EM5_JRdetectPV[0] )
   END_RUNG
   RUNG wire#w1
      Contact( "Unit1.Em5.ControlNodes".cmTransferPnPRightClampOpenClose.monitoring.inWorkPos )
      Contact( "Unit1.Em5.ControlNodes".transferPnPRight.sequence.status.seqActive )
      S_Coil( "Unit1.EmNodes".SpecialFunctionMode.EM5_JRdetectPV[2] )
   END_RUNG
   RUNG wire#w1
      Contact( "Unit1.Em5.ControlNodes".cmTransferPnPRightClampOpenClose.monitoring.inHomePos )
      Contact( "Unit1.Em5.ControlNodes".transferPnPRight.sequence.status.seqActive )
      wire#w3
      R_Coil( "Unit1.EmNodes".SpecialFunctionMode.EM5_JRdetectPV[2] )
   END_RUNG
   RUNG wire#w1
      Contact( "Unit1.EmNodes".unitStatus.state.stopped )
   END_RUNG wire#w3
   RUNG wire#w1
      Contact( "Unit1.EmNodes".SpecialFunctionMode.EM5_JRdetectPV[2] )
      Coil( "Unit1.EmNodes".SpecialFunctionMode.EM5_JRdetectPV[10] )
   END_RUNG
   RUNG wire#powerrail
      Contact( "Unit1.EmNodes".unitStatus.specialFunctions."Dry Run" )
      wire#w4
      Coil( "Unit1.Em5.Config".cmTransferPnPLeftClampOpenClose.disableFeedbackHomePos )
      Coil( "Unit1.Em5.Config".cmTransferPnPLeftClampOpenClose.disableFeedbackWorkPos )
      Coil( "Unit1.Em5.Config".cmTransferPnPLeftClampOpenClose.disableAlarms )
   END_RUNG
   RUNG wire#w4
      Coil( "Unit1.Em5.Config".cmTransferPnPRightClampOpenClose.disableFeedbackHomePos )
      Coil( "Unit1.Em5.Config".cmTransferPnPRightClampOpenClose.disableFeedbackWorkPos )
      Coil( "Unit1.Em5.Config".cmTransferPnPRightClampOpenClose.disableAlarms )
   END_RUNG
   // the same network as SCL:
   IF "Unit1.EmNodes".unitStatus.specialFunctions."Dry Run" AND "Unit1.Em5.ControlNodes".cmTransferPnPLeftClampOpenClose.monitoring.inWorkPos AND "Unit1.Em5.ControlNodes".transferPnPLeft.sequence.status.seqActive THEN
       "Unit1.EmNodes".SpecialFunctionMode.EM5_JRdetectPV[1] := TRUE;
   END_IF;
   IF "Unit1.EmNodes".unitStatus.specialFunctions."Dry Run" AND (("Unit1.Em5.ControlNodes".cmTransferPnPLeftClampOpenClose.monitoring.inHomePos AND "Unit1.Em5.ControlNodes".transferPnPLeft.sequence.status.seqActive) OR "Unit1.EmNodes".unitStatus.state.stopped) THEN
       "Unit1.EmNodes".SpecialFunctionMode.EM5_JRdetectPV[1] := FALSE;
   END_IF;
   "Unit1.EmNodes".SpecialFunctionMode.EM5_JRdetectPV[0] := "Unit1.EmNodes".unitStatus.specialFunctions."Dry Run" AND "Unit1.EmNodes".SpecialFunctionMode.EM5_JRdetectPV[1];
   IF "Unit1.EmNodes".unitStatus.specialFunctions."Dry Run" AND "Unit1.Em5.ControlNodes".cmTransferPnPRightClampOpenClose.monitoring.inWorkPos AND "Unit1.Em5.ControlNodes".transferPnPRight.sequence.status.seqActive THEN
       "Unit1.EmNodes".SpecialFunctionMode.EM5_JRdetectPV[2] := TRUE;
   END_IF;
   IF "Unit1.EmNodes".unitStatus.specialFunctions."Dry Run" AND (("Unit1.Em5.ControlNodes".cmTransferPnPRightClampOpenClose.monitoring.inHomePos AND "Unit1.Em5.ControlNodes".transferPnPRight.sequence.status.seqActive) OR "Unit1.EmNodes".unitStatus.state.stopped) THEN
       "Unit1.EmNodes".SpecialFunctionMode.EM5_JRdetectPV[2] := FALSE;
   END_IF;
   "Unit1.EmNodes".SpecialFunctionMode.EM5_JRdetectPV[10] := "Unit1.EmNodes".unitStatus.specialFunctions."Dry Run" AND "Unit1.EmNodes".SpecialFunctionMode.EM5_JRdetectPV[2];
   "Unit1.Em5.Config".cmTransferPnPLeftClampOpenClose.disableFeedbackHomePos := "Unit1.EmNodes".unitStatus.specialFunctions."Dry Run";
   "Unit1.Em5.Config".cmTransferPnPLeftClampOpenClose.disableFeedbackWorkPos := "Unit1.EmNodes".unitStatus.specialFunctions."Dry Run";
   "Unit1.Em5.Config".cmTransferPnPLeftClampOpenClose.disableAlarms := "Unit1.EmNodes".unitStatus.specialFunctions."Dry Run";
   "Unit1.Em5.Config".cmTransferPnPRightClampOpenClose.disableFeedbackHomePos := "Unit1.EmNodes".unitStatus.specialFunctions."Dry Run";
   "Unit1.Em5.Config".cmTransferPnPRightClampOpenClose.disableFeedbackWorkPos := "Unit1.EmNodes".unitStatus.specialFunctions."Dry Run";
   "Unit1.Em5.Config".cmTransferPnPRightClampOpenClose.disableAlarms := "Unit1.EmNodes".unitStatus.specialFunctions."Dry Run";
END_REGION

REGION Network 25: Transfer P&P Left & Right part detection data
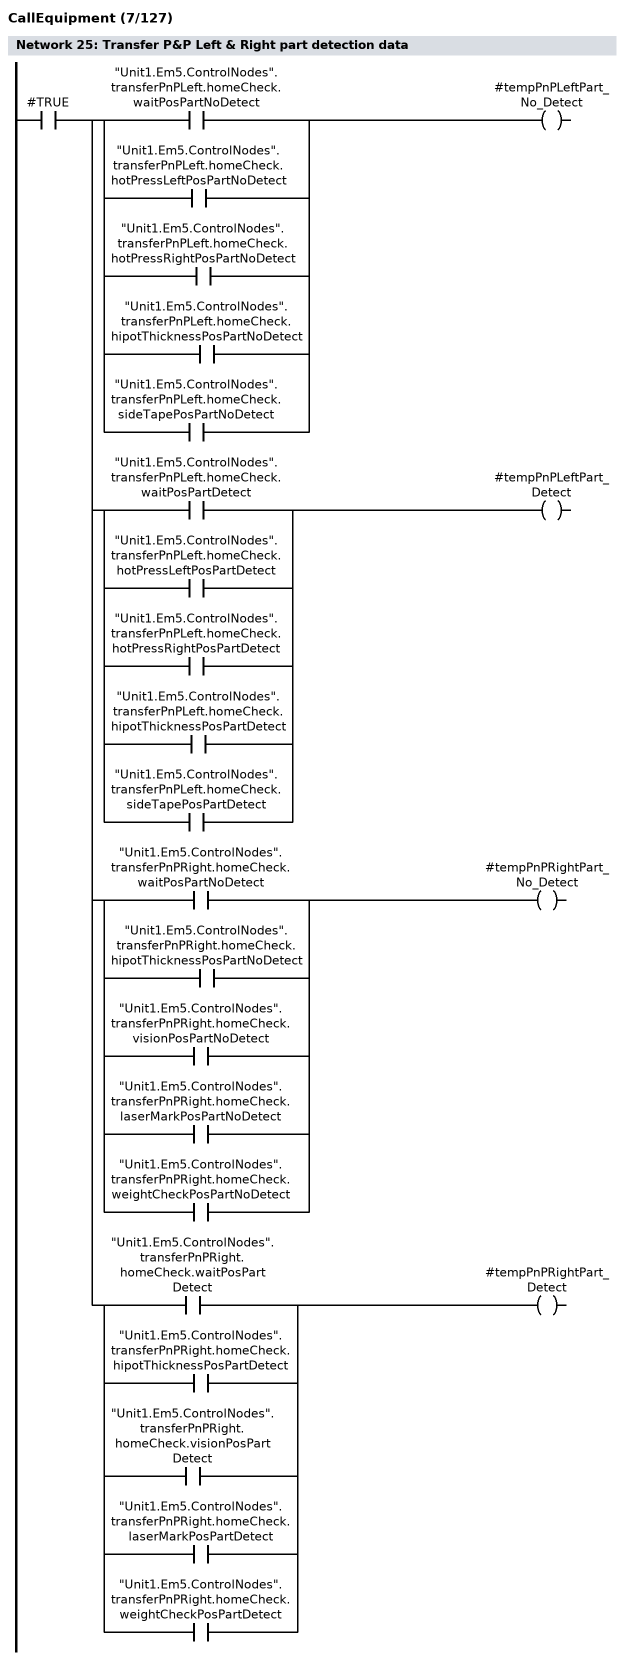
   RUNG wire#powerrail
      Contact( #TRUE )
      wire#w1
      Contact( "Unit1.Em5.ControlNodes".transferPnPLeft.homeCheck.waitPosPartNoDetect )
      wire#w2
      Coil( #tempPnPLeftPart_No_Detect )
   END_RUNG
   RUNG wire#w1
      Contact( "Unit1.Em5.ControlNodes".transferPnPLeft.homeCheck.hotPressLeftPosPartNoDetect )
   END_RUNG wire#w2
   RUNG wire#w1
      Contact( "Unit1.Em5.ControlNodes".transferPnPLeft.homeCheck.hotPressRightPosPartNoDetect )
   END_RUNG wire#w2
   RUNG wire#w1
      Contact( "Unit1.Em5.ControlNodes".transferPnPLeft.homeCheck.hipotThicknessPosPartNoDetect )
   END_RUNG wire#w2
   RUNG wire#w1
      Contact( "Unit1.Em5.ControlNodes".transferPnPLeft.homeCheck.sideTapePosPartNoDetect )
   END_RUNG wire#w2
   RUNG wire#w1
      Contact( "Unit1.Em5.ControlNodes".transferPnPLeft.homeCheck.waitPosPartDetect )
      wire#w3
      Coil( #tempPnPLeftPart_Detect )
   END_RUNG
   RUNG wire#w1
      Contact( "Unit1.Em5.ControlNodes".transferPnPLeft.homeCheck.hotPressLeftPosPartDetect )
   END_RUNG wire#w3
   RUNG wire#w1
      Contact( "Unit1.Em5.ControlNodes".transferPnPLeft.homeCheck.hotPressRightPosPartDetect )
   END_RUNG wire#w3
   RUNG wire#w1
      Contact( "Unit1.Em5.ControlNodes".transferPnPLeft.homeCheck.hipotThicknessPosPartDetect )
   END_RUNG wire#w3
   RUNG wire#w1
      Contact( "Unit1.Em5.ControlNodes".transferPnPLeft.homeCheck.sideTapePosPartDetect )
   END_RUNG wire#w3
   RUNG wire#w1
      Contact( "Unit1.Em5.ControlNodes".transferPnPRight.homeCheck.waitPosPartNoDetect )
      wire#w4
      Coil( #tempPnPRightPart_No_Detect )
   END_RUNG
   RUNG wire#w1
      Contact( "Unit1.Em5.ControlNodes".transferPnPRight.homeCheck.hipotThicknessPosPartNoDetect )
   END_RUNG wire#w4
   RUNG wire#w1
      Contact( "Unit1.Em5.ControlNodes".transferPnPRight.homeCheck.visionPosPartNoDetect )
   END_RUNG wire#w4
   RUNG wire#w1
      Contact( "Unit1.Em5.ControlNodes".transferPnPRight.homeCheck.laserMarkPosPartNoDetect )
   END_RUNG wire#w4
   RUNG wire#w1
      Contact( "Unit1.Em5.ControlNodes".transferPnPRight.homeCheck.weightCheckPosPartNoDetect )
   END_RUNG wire#w4
   RUNG wire#w1
      Contact( "Unit1.Em5.ControlNodes".transferPnPRight.homeCheck.waitPosPartDetect )
      wire#w5
      Coil( #tempPnPRightPart_Detect )
   END_RUNG
   RUNG wire#w1
      Contact( "Unit1.Em5.ControlNodes".transferPnPRight.homeCheck.hipotThicknessPosPartDetect )
   END_RUNG wire#w5
   RUNG wire#w1
      Contact( "Unit1.Em5.ControlNodes".transferPnPRight.homeCheck.visionPosPartDetect )
   END_RUNG wire#w5
   RUNG wire#w1
      Contact( "Unit1.Em5.ControlNodes".transferPnPRight.homeCheck.laserMarkPosPartDetect )
   END_RUNG wire#w5
   RUNG wire#w1
      Contact( "Unit1.Em5.ControlNodes".transferPnPRight.homeCheck.weightCheckPosPartDetect )
   END_RUNG wire#w5
   // the same network as SCL:
   #tempPnPLeftPart_No_Detect := #TRUE AND ("Unit1.Em5.ControlNodes".transferPnPLeft.homeCheck.waitPosPartNoDetect OR "Unit1.Em5.ControlNodes".transferPnPLeft.homeCheck.hotPressLeftPosPartNoDetect OR "Unit1.Em5.ControlNodes".transferPnPLeft.homeCheck.hotPressRightPosPartNoDetect OR "Unit1.Em5.ControlNodes".transferPnPLeft.homeCheck.hipotThicknessPosPartNoDetect OR "Unit1.Em5.ControlNodes".transferPnPLeft.homeCheck.sideTapePosPartNoDetect);
   #tempPnPLeftPart_Detect := #TRUE AND ("Unit1.Em5.ControlNodes".transferPnPLeft.homeCheck.waitPosPartDetect OR "Unit1.Em5.ControlNodes".transferPnPLeft.homeCheck.hotPressLeftPosPartDetect OR "Unit1.Em5.ControlNodes".transferPnPLeft.homeCheck.hotPressRightPosPartDetect OR "Unit1.Em5.ControlNodes".transferPnPLeft.homeCheck.hipotThicknessPosPartDetect OR "Unit1.Em5.ControlNodes".transferPnPLeft.homeCheck.sideTapePosPartDetect);
   #tempPnPRightPart_No_Detect := #TRUE AND ("Unit1.Em5.ControlNodes".transferPnPRight.homeCheck.waitPosPartNoDetect OR "Unit1.Em5.ControlNodes".transferPnPRight.homeCheck.hipotThicknessPosPartNoDetect OR "Unit1.Em5.ControlNodes".transferPnPRight.homeCheck.visionPosPartNoDetect OR "Unit1.Em5.ControlNodes".transferPnPRight.homeCheck.laserMarkPosPartNoDetect OR "Unit1.Em5.ControlNodes".transferPnPRight.homeCheck.weightCheckPosPartNoDetect);
   #tempPnPRightPart_Detect := #TRUE AND ("Unit1.Em5.ControlNodes".transferPnPRight.homeCheck.waitPosPartDetect OR "Unit1.Em5.ControlNodes".transferPnPRight.homeCheck.hipotThicknessPosPartDetect OR "Unit1.Em5.ControlNodes".transferPnPRight.homeCheck.visionPosPartDetect OR "Unit1.Em5.ControlNodes".transferPnPRight.homeCheck.laserMarkPosPartDetect OR "Unit1.Em5.ControlNodes".transferPnPRight.homeCheck.weightCheckPosPartDetect);
END_REGION

REGION Network 27: [Job]Transfer P&P Left Select Job [initializing]
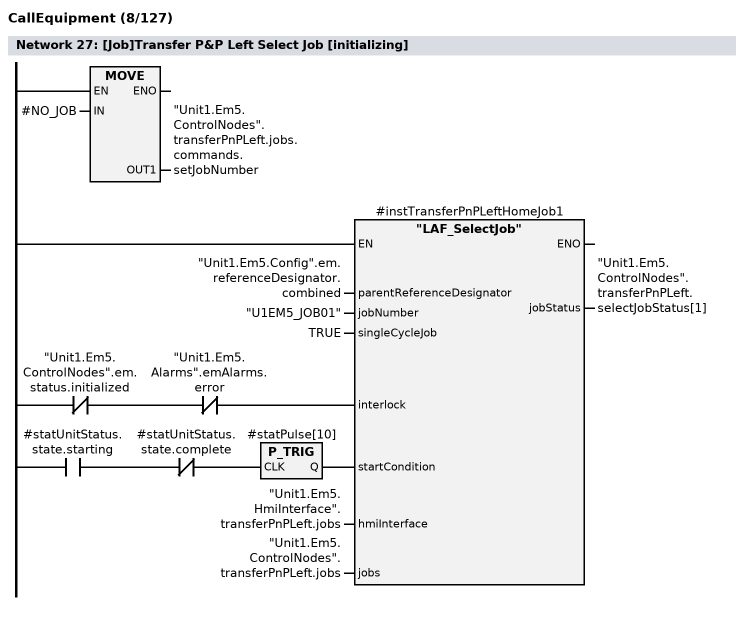
   RUNG wire#powerrail
      Move(in := #NO_JOB, out1 => "Unit1.Em5.ControlNodes".transferPnPLeft.jobs.commands.setJobNumber)
   END_RUNG
   RUNG wire#powerrail
      #instTransferPnPLeftHomeJob1(interlock := wire#w1, startCondition := wire#w2, parentReferenceDesignator := "Unit1.Em5.Config".em.referenceDesignator.combined, jobNumber := "U1EM5_JOB01", singleCycleJob := TRUE, hmiInterface := "Unit1.Em5.HmiInterface".transferPnPLeft.jobs, jobs := "Unit1.Em5.ControlNodes".transferPnPLeft.jobs, jobStatus => "Unit1.Em5.ControlNodes".transferPnPLeft.selectJobStatus[1])
   END_RUNG
   RUNG wire#powerrail
      I_Contact( "Unit1.Em5.ControlNodes".em.status.initialized )
      I_Contact( "Unit1.Em5.Alarms".emAlarms.error )
   END_RUNG wire#w1
   RUNG wire#powerrail
      Contact( #statUnitStatus.state.starting )
      I_Contact( #statUnitStatus.state.complete )
      P_Trig( #statPulse[10] )
   END_RUNG wire#w2
   // the same network as SCL:
   "Unit1.Em5.ControlNodes".transferPnPLeft.jobs.commands.setJobNumber := #NO_JOB;
   #_w1 := #statUnitStatus.state.starting AND NOT #statUnitStatus.state.complete;
   #_w2 := #_w1 AND NOT #statPulse[10];   // rising edge
   #statPulse[10] := #_w1;
   #instTransferPnPLeftHomeJob1(parentReferenceDesignator := "Unit1.Em5.Config".em.referenceDesignator.combined,   // "LAF_SelectJob"
                           jobNumber := "U1EM5_JOB01",
                           singleCycleJob := TRUE,
                           interlock := NOT "Unit1.Em5.ControlNodes".em.status.initialized AND NOT "Unit1.Em5.Alarms".emAlarms.error,
                           startCondition := #_w2,
                           hmiInterface := "Unit1.Em5.HmiInterface".transferPnPLeft.jobs,
                           jobs := "Unit1.Em5.ControlNodes".transferPnPLeft.jobs,
                           jobStatus => "Unit1.Em5.ControlNodes".transferPnPLeft.selectJobStatus[1]);
END_REGION

REGION Network 28: [Job]Transfer P&P Left Select Job [BA30 - A]
   // Configure here when the jobs of the sequence should be started. More jobs could be added.
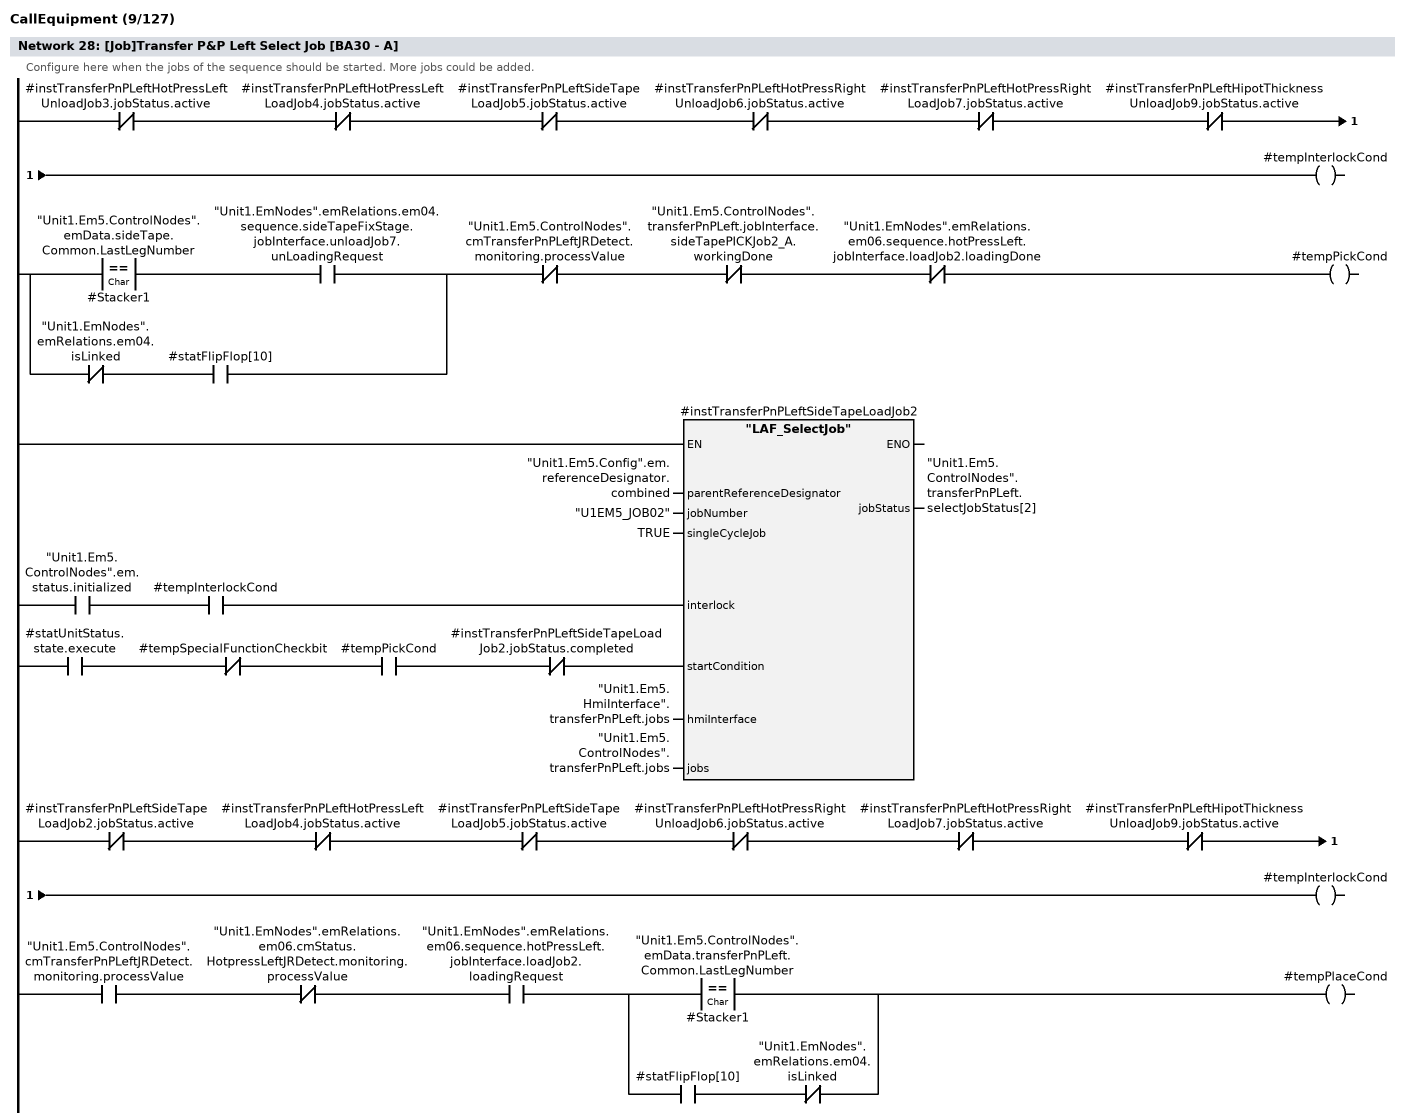
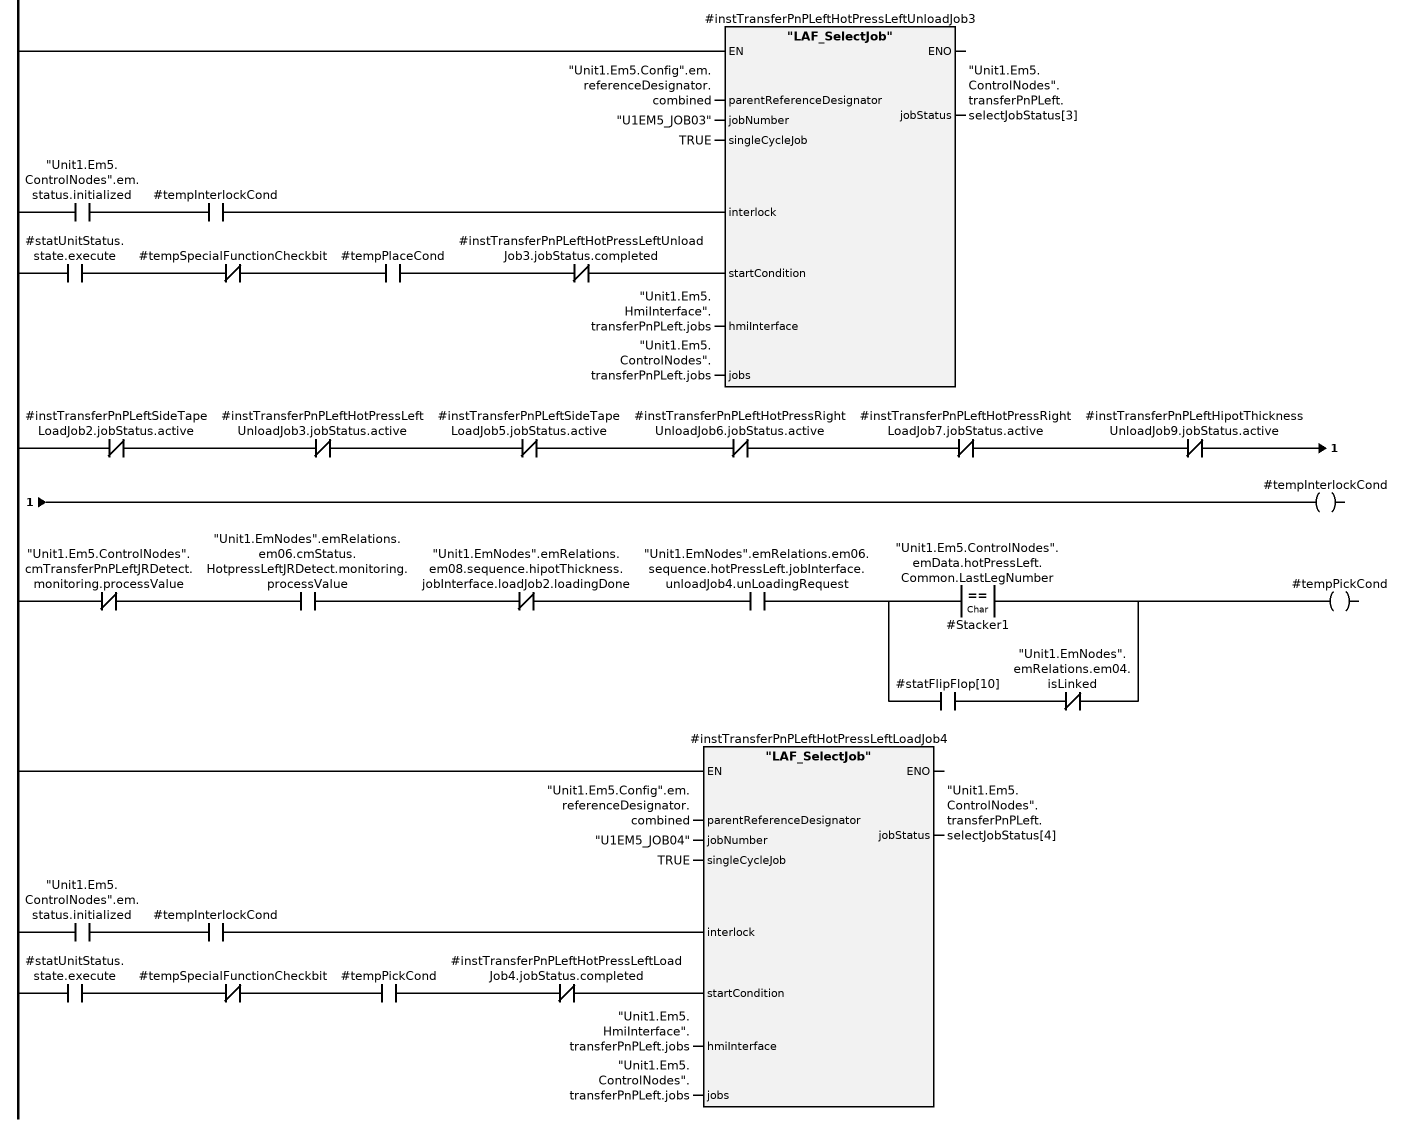
   RUNG wire#powerrail
      I_Contact( #instTransferPnPLeftHotPressLeftUnloadJob3.jobStatus.active )
      I_Contact( #instTransferPnPLeftHotPressLeftLoadJob4.jobStatus.active )
      I_Contact( #instTransferPnPLeftSideTapeLoadJob5.jobStatus.active )
      I_Contact( #instTransferPnPLeftHotPressRightUnloadJob6.jobStatus.active )
      I_Contact( #instTransferPnPLeftHotPressRightLoadJob7.jobStatus.active )
      I_Contact( #instTransferPnPLeftHipotThicknessUnloadJob9.jobStatus.active )
      Coil( #tempInterlockCond )
   END_RUNG
   RUNG wire#powerrail
      { S7_Templates := "SrcType := Char" } EQ_Contact(in1 := "Unit1.Em5.ControlNodes".emData.sideTape.Common.LastLegNumber, in2 := #Stacker1)
      Contact( "Unit1.EmNodes".emRelations.em04.sequence.sideTapeFixStage.jobInterface.unloadJob7.unLoadingRequest )
      wire#w1
      I_Contact( "Unit1.Em5.ControlNodes".cmTransferPnPLeftJRDetect.monitoring.processValue )
      I_Contact( "Unit1.Em5.ControlNodes".transferPnPLeft.jobInterface.sideTapePICKJob2_A.workingDone )
      I_Contact( "Unit1.EmNodes".emRelations.em06.sequence.hotPressLeft.jobInterface.loadJob2.loadingDone )
      Coil( #tempPickCond )
   END_RUNG
   RUNG wire#powerrail
      I_Contact( "Unit1.EmNodes".emRelations.em04.isLinked )
      Contact( #statFlipFlop[10] )
   END_RUNG wire#w1
   RUNG wire#powerrail
      #instTransferPnPLeftSideTapeLoadJob2(interlock := wire#w2, startCondition := wire#w3, parentReferenceDesignator := "Unit1.Em5.Config".em.referenceDesignator.combined, jobNumber := "U1EM5_JOB02", singleCycleJob := TRUE, hmiInterface := "Unit1.Em5.HmiInterface".transferPnPLeft.jobs, jobs := "Unit1.Em5.ControlNodes".transferPnPLeft.jobs, jobStatus => "Unit1.Em5.ControlNodes".transferPnPLeft.selectJobStatus[2])
   END_RUNG
   RUNG wire#powerrail
      Contact( "Unit1.Em5.ControlNodes".em.status.initialized )
      Contact( #tempInterlockCond )
   END_RUNG wire#w2
   RUNG wire#powerrail
      Contact( #statUnitStatus.state.execute )
      I_Contact( #tempSpecialFunctionCheckbit )
      Contact( #tempPickCond )
      I_Contact( #instTransferPnPLeftSideTapeLoadJob2.jobStatus.completed )
   END_RUNG wire#w3
   RUNG wire#powerrail
      I_Contact( #instTransferPnPLeftSideTapeLoadJob2.jobStatus.active )
      I_Contact( #instTransferPnPLeftHotPressLeftLoadJob4.jobStatus.active )
      I_Contact( #instTransferPnPLeftSideTapeLoadJob5.jobStatus.active )
      I_Contact( #instTransferPnPLeftHotPressRightUnloadJob6.jobStatus.active )
      I_Contact( #instTransferPnPLeftHotPressRightLoadJob7.jobStatus.active )
      I_Contact( #instTransferPnPLeftHipotThicknessUnloadJob9.jobStatus.active )
      Coil( #tempInterlockCond )
   END_RUNG
   RUNG wire#powerrail
      Contact( "Unit1.Em5.ControlNodes".cmTransferPnPLeftJRDetect.monitoring.processValue )
      I_Contact( "Unit1.EmNodes".emRelations.em06.cmStatus.HotpressLeftJRDetect.monitoring.processValue )
      Contact( "Unit1.EmNodes".emRelations.em06.sequence.hotPressLeft.jobInterface.loadJob2.loadingRequest )
      wire#w4
      { S7_Templates := "SrcType := Char" } EQ_Contact(in1 := "Unit1.Em5.ControlNodes".emData.transferPnPLeft.Common.LastLegNumber, in2 := #Stacker1)
      wire#w5
      Coil( #tempPlaceCond )
   END_RUNG
   RUNG wire#w4
      Contact( #statFlipFlop[10] )
      I_Contact( "Unit1.EmNodes".emRelations.em04.isLinked )
   END_RUNG wire#w5
   RUNG wire#powerrail
      #instTransferPnPLeftHotPressLeftUnloadJob3(interlock := wire#w6, startCondition := wire#w7, parentReferenceDesignator := "Unit1.Em5.Config".em.referenceDesignator.combined, jobNumber := "U1EM5_JOB03", singleCycleJob := TRUE, hmiInterface := "Unit1.Em5.HmiInterface".transferPnPLeft.jobs, jobs := "Unit1.Em5.ControlNodes".transferPnPLeft.jobs, jobStatus => "Unit1.Em5.ControlNodes".transferPnPLeft.selectJobStatus[3])
   END_RUNG
   RUNG wire#powerrail
      Contact( "Unit1.Em5.ControlNodes".em.status.initialized )
      Contact( #tempInterlockCond )
   END_RUNG wire#w6
   RUNG wire#powerrail
      Contact( #statUnitStatus.state.execute )
      I_Contact( #tempSpecialFunctionCheckbit )
      Contact( #tempPlaceCond )
      I_Contact( #instTransferPnPLeftHotPressLeftUnloadJob3.jobStatus.completed )
   END_RUNG wire#w7
   RUNG wire#powerrail
      I_Contact( #instTransferPnPLeftSideTapeLoadJob2.jobStatus.active )
      I_Contact( #instTransferPnPLeftHotPressLeftUnloadJob3.jobStatus.active )
      I_Contact( #instTransferPnPLeftSideTapeLoadJob5.jobStatus.active )
      I_Contact( #instTransferPnPLeftHotPressRightUnloadJob6.jobStatus.active )
      I_Contact( #instTransferPnPLeftHotPressRightLoadJob7.jobStatus.active )
      I_Contact( #instTransferPnPLeftHipotThicknessUnloadJob9.jobStatus.active )
      Coil( #tempInterlockCond )
   END_RUNG
   RUNG wire#powerrail
      I_Contact( "Unit1.Em5.ControlNodes".cmTransferPnPLeftJRDetect.monitoring.processValue )
      Contact( "Unit1.EmNodes".emRelations.em06.cmStatus.HotpressLeftJRDetect.monitoring.processValue )
      I_Contact( "Unit1.EmNodes".emRelations.em08.sequence.hipotThickness.jobInterface.loadJob2.loadingDone )
      Contact( "Unit1.EmNodes".emRelations.em06.sequence.hotPressLeft.jobInterface.unloadJob4.unLoadingRequest )
      wire#w8
      { S7_Templates := "SrcType := Char" } EQ_Contact(in1 := "Unit1.Em5.ControlNodes".emData.hotPressLeft.Common.LastLegNumber, in2 := #Stacker1)
      wire#w9
      Coil( #tempPickCond )
   END_RUNG
   RUNG wire#w8
      Contact( #statFlipFlop[10] )
      I_Contact( "Unit1.EmNodes".emRelations.em04.isLinked )
   END_RUNG wire#w9
   RUNG wire#powerrail
      #instTransferPnPLeftHotPressLeftLoadJob4(interlock := wire#w10, startCondition := wire#w11, parentReferenceDesignator := "Unit1.Em5.Config".em.referenceDesignator.combined, jobNumber := "U1EM5_JOB04", singleCycleJob := TRUE, hmiInterface := "Unit1.Em5.HmiInterface".transferPnPLeft.jobs, jobs := "Unit1.Em5.ControlNodes".transferPnPLeft.jobs, jobStatus => "Unit1.Em5.ControlNodes".transferPnPLeft.selectJobStatus[4])
   END_RUNG
   RUNG wire#powerrail
      Contact( "Unit1.Em5.ControlNodes".em.status.initialized )
      Contact( #tempInterlockCond )
   END_RUNG wire#w10
   RUNG wire#powerrail
      Contact( #statUnitStatus.state.execute )
      I_Contact( #tempSpecialFunctionCheckbit )
      Contact( #tempPickCond )
      I_Contact( #instTransferPnPLeftHotPressLeftLoadJob4.jobStatus.completed )
   END_RUNG wire#w11
   // the same network as SCL:
   #tempInterlockCond := NOT #instTransferPnPLeftHotPressLeftUnloadJob3.jobStatus.active AND NOT #instTransferPnPLeftHotPressLeftLoadJob4.jobStatus.active AND NOT #instTransferPnPLeftSideTapeLoadJob5.jobStatus.active AND NOT #instTransferPnPLeftHotPressRightUnloadJob6.jobStatus.active AND NOT #instTransferPnPLeftHotPressRightLoadJob7.jobStatus.active AND NOT #instTransferPnPLeftHipotThicknessUnloadJob9.jobStatus.active;
   #tempPickCond := ((("Unit1.Em5.ControlNodes".emData.sideTape.Common.LastLegNumber = #Stacker1) AND "Unit1.EmNodes".emRelations.em04.sequence.sideTapeFixStage.jobInterface.unloadJob7.unLoadingRequest) OR (NOT "Unit1.EmNodes".emRelations.em04.isLinked AND #statFlipFlop[10])) AND NOT "Unit1.Em5.ControlNodes".cmTransferPnPLeftJRDetect.monitoring.processValue AND NOT "Unit1.Em5.ControlNodes".transferPnPLeft.jobInterface.sideTapePICKJob2_A.workingDone AND NOT "Unit1.EmNodes".emRelations.em06.sequence.hotPressLeft.jobInterface.loadJob2.loadingDone;
   #instTransferPnPLeftSideTapeLoadJob2(parentReferenceDesignator := "Unit1.Em5.Config".em.referenceDesignator.combined,   // "LAF_SelectJob"
                           jobNumber := "U1EM5_JOB02",
                           singleCycleJob := TRUE,
                           interlock := "Unit1.Em5.ControlNodes".em.status.initialized AND #tempInterlockCond,
                           startCondition := #statUnitStatus.state.execute AND NOT #tempSpecialFunctionCheckbit AND #tempPickCond AND NOT #instTransferPnPLeftSideTapeLoadJob2.jobStatus.completed,
                           hmiInterface := "Unit1.Em5.HmiInterface".transferPnPLeft.jobs,
                           jobs := "Unit1.Em5.ControlNodes".transferPnPLeft.jobs,
                           jobStatus => "Unit1.Em5.ControlNodes".transferPnPLeft.selectJobStatus[2]);
   #tempInterlockCond := NOT #instTransferPnPLeftSideTapeLoadJob2.jobStatus.active AND NOT #instTransferPnPLeftHotPressLeftLoadJob4.jobStatus.active AND NOT #instTransferPnPLeftSideTapeLoadJob5.jobStatus.active AND NOT #instTransferPnPLeftHotPressRightUnloadJob6.jobStatus.active AND NOT #instTransferPnPLeftHotPressRightLoadJob7.jobStatus.active AND NOT #instTransferPnPLeftHipotThicknessUnloadJob9.jobStatus.active;
   #tempPlaceCond := "Unit1.Em5.ControlNodes".cmTransferPnPLeftJRDetect.monitoring.processValue AND NOT "Unit1.EmNodes".emRelations.em06.cmStatus.HotpressLeftJRDetect.monitoring.processValue AND "Unit1.EmNodes".emRelations.em06.sequence.hotPressLeft.jobInterface.loadJob2.loadingRequest AND (("Unit1.Em5.ControlNodes".emData.transferPnPLeft.Common.LastLegNumber = #Stacker1) OR (#statFlipFlop[10] AND NOT "Unit1.EmNodes".emRelations.em04.isLinked));
   #instTransferPnPLeftHotPressLeftUnloadJob3(parentReferenceDesignator := "Unit1.Em5.Config".em.referenceDesignator.combined,   // "LAF_SelectJob"
                           jobNumber := "U1EM5_JOB03",
                           singleCycleJob := TRUE,
                           interlock := "Unit1.Em5.ControlNodes".em.status.initialized AND #tempInterlockCond,
                           startCondition := #statUnitStatus.state.execute AND NOT #tempSpecialFunctionCheckbit AND #tempPlaceCond AND NOT #instTransferPnPLeftHotPressLeftUnloadJob3.jobStatus.completed,
                           hmiInterface := "Unit1.Em5.HmiInterface".transferPnPLeft.jobs,
                           jobs := "Unit1.Em5.ControlNodes".transferPnPLeft.jobs,
                           jobStatus => "Unit1.Em5.ControlNodes".transferPnPLeft.selectJobStatus[3]);
   #tempInterlockCond := NOT #instTransferPnPLeftSideTapeLoadJob2.jobStatus.active AND NOT #instTransferPnPLeftHotPressLeftUnloadJob3.jobStatus.active AND NOT #instTransferPnPLeftSideTapeLoadJob5.jobStatus.active AND NOT #instTransferPnPLeftHotPressRightUnloadJob6.jobStatus.active AND NOT #instTransferPnPLeftHotPressRightLoadJob7.jobStatus.active AND NOT #instTransferPnPLeftHipotThicknessUnloadJob9.jobStatus.active;
   #tempPickCond := NOT "Unit1.Em5.ControlNodes".cmTransferPnPLeftJRDetect.monitoring.processValue AND "Unit1.EmNodes".emRelations.em06.cmStatus.HotpressLeftJRDetect.monitoring.processValue AND NOT "Unit1.EmNodes".emRelations.em08.sequence.hipotThickness.jobInterface.loadJob2.loadingDone AND "Unit1.EmNodes".emRelations.em06.sequence.hotPressLeft.jobInterface.unloadJob4.unLoadingRequest AND (("Unit1.Em5.ControlNodes".emData.hotPressLeft.Common.LastLegNumber = #Stacker1) OR (#statFlipFlop[10] AND NOT "Unit1.EmNodes".emRelations.em04.isLinked));
   #instTransferPnPLeftHotPressLeftLoadJob4(parentReferenceDesignator := "Unit1.Em5.Config".em.referenceDesignator.combined,   // "LAF_SelectJob"
                           jobNumber := "U1EM5_JOB04",
                           singleCycleJob := TRUE,
                           interlock := "Unit1.Em5.ControlNodes".em.status.initialized AND #tempInterlockCond,
                           startCondition := #statUnitStatus.state.execute AND NOT #tempSpecialFunctionCheckbit AND #tempPickCond AND NOT #instTransferPnPLeftHotPressLeftLoadJob4.jobStatus.completed,
                           hmiInterface := "Unit1.Em5.HmiInterface".transferPnPLeft.jobs,
                           jobs := "Unit1.Em5.ControlNodes".transferPnPLeft.jobs,
                           jobStatus => "Unit1.Em5.ControlNodes".transferPnPLeft.selectJobStatus[4]);
END_REGION

REGION Network 29: Transfer P&P Left Job Interface [Side Tape Loading][A]
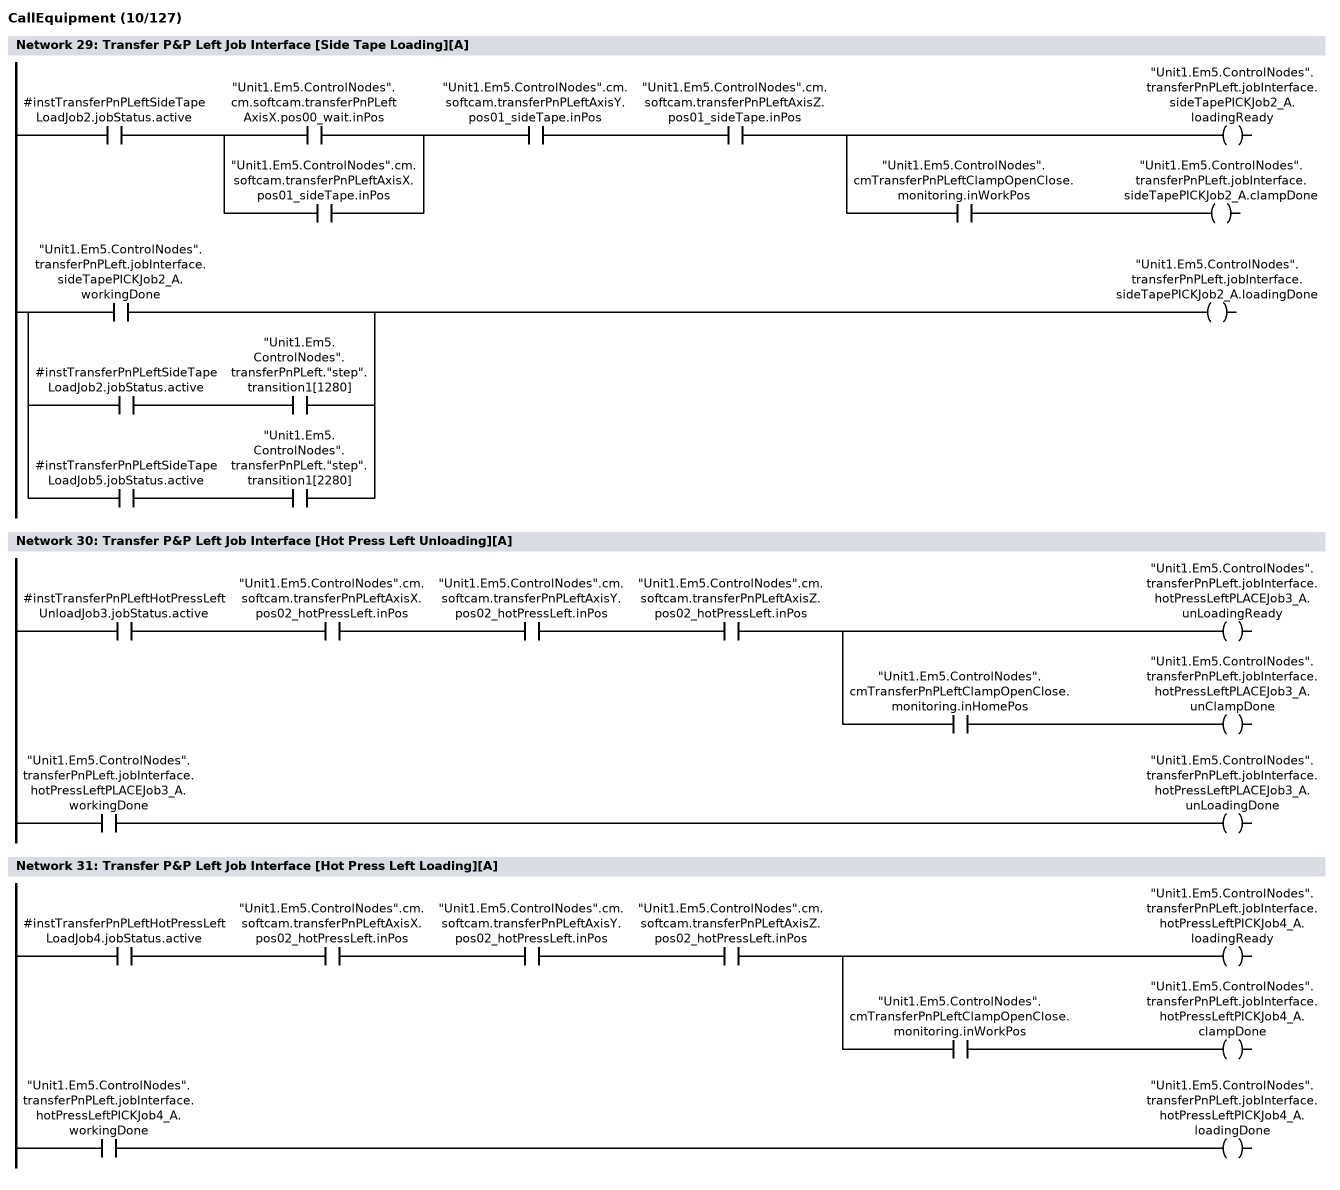
   RUNG wire#powerrail
      Contact( #instTransferPnPLeftSideTapeLoadJob2.jobStatus.active )
      wire#w1
      Contact( "Unit1.Em5.ControlNodes".cm.softcam.transferPnPLeftAxisX.pos00_wait.inPos )
      wire#w2
      Contact( "Unit1.Em5.ControlNodes".cm.softcam.transferPnPLeftAxisY.pos01_sideTape.inPos )
      Contact( "Unit1.Em5.ControlNodes".cm.softcam.transferPnPLeftAxisZ.pos01_sideTape.inPos )
      wire#w3
      Coil( "Unit1.Em5.ControlNodes".transferPnPLeft.jobInterface.sideTapePICKJob2_A.loadingReady )
   END_RUNG
   RUNG wire#w1
      Contact( "Unit1.Em5.ControlNodes".cm.softcam.transferPnPLeftAxisX.pos01_sideTape.inPos )
   END_RUNG wire#w2
   RUNG wire#w3
      Contact( "Unit1.Em5.ControlNodes".cmTransferPnPLeftClampOpenClose.monitoring.inWorkPos )
      Coil( "Unit1.Em5.ControlNodes".transferPnPLeft.jobInterface.sideTapePICKJob2_A.clampDone )
   END_RUNG
   RUNG wire#powerrail
      Contact( "Unit1.Em5.ControlNodes".transferPnPLeft.jobInterface.sideTapePICKJob2_A.workingDone )
      wire#w4
      Coil( "Unit1.Em5.ControlNodes".transferPnPLeft.jobInterface.sideTapePICKJob2_A.loadingDone )
   END_RUNG
   RUNG wire#powerrail
      Contact( #instTransferPnPLeftSideTapeLoadJob2.jobStatus.active )
      Contact( "Unit1.Em5.ControlNodes".transferPnPLeft."step".transition1[1280] )
   END_RUNG wire#w4
   RUNG wire#powerrail
      Contact( #instTransferPnPLeftSideTapeLoadJob5.jobStatus.active )
      Contact( "Unit1.Em5.ControlNodes".transferPnPLeft."step".transition1[2280] )
   END_RUNG wire#w4
   // the same network as SCL:
   "Unit1.Em5.ControlNodes".transferPnPLeft.jobInterface.sideTapePICKJob2_A.loadingReady := #instTransferPnPLeftSideTapeLoadJob2.jobStatus.active AND ("Unit1.Em5.ControlNodes".cm.softcam.transferPnPLeftAxisX.pos00_wait.inPos OR "Unit1.Em5.ControlNodes".cm.softcam.transferPnPLeftAxisX.pos01_sideTape.inPos) AND "Unit1.Em5.ControlNodes".cm.softcam.transferPnPLeftAxisY.pos01_sideTape.inPos AND "Unit1.Em5.ControlNodes".cm.softcam.transferPnPLeftAxisZ.pos01_sideTape.inPos;
   "Unit1.Em5.ControlNodes".transferPnPLeft.jobInterface.sideTapePICKJob2_A.clampDone := "Unit1.Em5.ControlNodes".transferPnPLeft.jobInterface.sideTapePICKJob2_A.loadingReady AND "Unit1.Em5.ControlNodes".cmTransferPnPLeftClampOpenClose.monitoring.inWorkPos;
   "Unit1.Em5.ControlNodes".transferPnPLeft.jobInterface.sideTapePICKJob2_A.loadingDone := "Unit1.Em5.ControlNodes".transferPnPLeft.jobInterface.sideTapePICKJob2_A.workingDone OR (#instTransferPnPLeftSideTapeLoadJob2.jobStatus.active AND "Unit1.Em5.ControlNodes".transferPnPLeft."step".transition1[1280]) OR (#instTransferPnPLeftSideTapeLoadJob5.jobStatus.active AND "Unit1.Em5.ControlNodes".transferPnPLeft."step".transition1[2280]);
END_REGION

REGION Network 30: Transfer P&P Left Job Interface [Hot Press Left Unloading][A]
   RUNG wire#powerrail
      Contact( #instTransferPnPLeftHotPressLeftUnloadJob3.jobStatus.active )
      Contact( "Unit1.Em5.ControlNodes".cm.softcam.transferPnPLeftAxisX.pos02_hotPressLeft.inPos )
      Contact( "Unit1.Em5.ControlNodes".cm.softcam.transferPnPLeftAxisY.pos02_hotPressLeft.inPos )
      Contact( "Unit1.Em5.ControlNodes".cm.softcam.transferPnPLeftAxisZ.pos02_hotPressLeft.inPos )
      wire#w1
      Coil( "Unit1.Em5.ControlNodes".transferPnPLeft.jobInterface.hotPressLeftPLACEJob3_A.unLoadingReady )
   END_RUNG
   RUNG wire#w1
      Contact( "Unit1.Em5.ControlNodes".cmTransferPnPLeftClampOpenClose.monitoring.inHomePos )
      Coil( "Unit1.Em5.ControlNodes".transferPnPLeft.jobInterface.hotPressLeftPLACEJob3_A.unClampDone )
   END_RUNG
   RUNG wire#powerrail
      Contact( "Unit1.Em5.ControlNodes".transferPnPLeft.jobInterface.hotPressLeftPLACEJob3_A.workingDone )
      Coil( "Unit1.Em5.ControlNodes".transferPnPLeft.jobInterface.hotPressLeftPLACEJob3_A.unLoadingDone )
   END_RUNG
   // the same network as SCL:
   "Unit1.Em5.ControlNodes".transferPnPLeft.jobInterface.hotPressLeftPLACEJob3_A.unLoadingReady := #instTransferPnPLeftHotPressLeftUnloadJob3.jobStatus.active AND "Unit1.Em5.ControlNodes".cm.softcam.transferPnPLeftAxisX.pos02_hotPressLeft.inPos AND "Unit1.Em5.ControlNodes".cm.softcam.transferPnPLeftAxisY.pos02_hotPressLeft.inPos AND "Unit1.Em5.ControlNodes".cm.softcam.transferPnPLeftAxisZ.pos02_hotPressLeft.inPos;
   "Unit1.Em5.ControlNodes".transferPnPLeft.jobInterface.hotPressLeftPLACEJob3_A.unClampDone := "Unit1.Em5.ControlNodes".transferPnPLeft.jobInterface.hotPressLeftPLACEJob3_A.unLoadingReady AND "Unit1.Em5.ControlNodes".cmTransferPnPLeftClampOpenClose.monitoring.inHomePos;
   "Unit1.Em5.ControlNodes".transferPnPLeft.jobInterface.hotPressLeftPLACEJob3_A.unLoadingDone := "Unit1.Em5.ControlNodes".transferPnPLeft.jobInterface.hotPressLeftPLACEJob3_A.workingDone;
END_REGION

REGION Network 31: Transfer P&P Left Job Interface [Hot Press Left Loading][A]
   RUNG wire#powerrail
      Contact( #instTransferPnPLeftHotPressLeftLoadJob4.jobStatus.active )
      Contact( "Unit1.Em5.ControlNodes".cm.softcam.transferPnPLeftAxisX.pos02_hotPressLeft.inPos )
      Contact( "Unit1.Em5.ControlNodes".cm.softcam.transferPnPLeftAxisY.pos02_hotPressLeft.inPos )
      Contact( "Unit1.Em5.ControlNodes".cm.softcam.transferPnPLeftAxisZ.pos02_hotPressLeft.inPos )
      wire#w1
      Coil( "Unit1.Em5.ControlNodes".transferPnPLeft.jobInterface.hotPressLeftPICKJob4_A.loadingReady )
   END_RUNG
   RUNG wire#w1
      Contact( "Unit1.Em5.ControlNodes".cmTransferPnPLeftClampOpenClose.monitoring.inWorkPos )
      Coil( "Unit1.Em5.ControlNodes".transferPnPLeft.jobInterface.hotPressLeftPICKJob4_A.clampDone )
   END_RUNG
   RUNG wire#powerrail
      Contact( "Unit1.Em5.ControlNodes".transferPnPLeft.jobInterface.hotPressLeftPICKJob4_A.workingDone )
      Coil( "Unit1.Em5.ControlNodes".transferPnPLeft.jobInterface.hotPressLeftPICKJob4_A.loadingDone )
   END_RUNG
   // the same network as SCL:
   "Unit1.Em5.ControlNodes".transferPnPLeft.jobInterface.hotPressLeftPICKJob4_A.loadingReady := #instTransferPnPLeftHotPressLeftLoadJob4.jobStatus.active AND "Unit1.Em5.ControlNodes".cm.softcam.transferPnPLeftAxisX.pos02_hotPressLeft.inPos AND "Unit1.Em5.ControlNodes".cm.softcam.transferPnPLeftAxisY.pos02_hotPressLeft.inPos AND "Unit1.Em5.ControlNodes".cm.softcam.transferPnPLeftAxisZ.pos02_hotPressLeft.inPos;
   "Unit1.Em5.ControlNodes".transferPnPLeft.jobInterface.hotPressLeftPICKJob4_A.clampDone := "Unit1.Em5.ControlNodes".transferPnPLeft.jobInterface.hotPressLeftPICKJob4_A.loadingReady AND "Unit1.Em5.ControlNodes".cmTransferPnPLeftClampOpenClose.monitoring.inWorkPos;
   "Unit1.Em5.ControlNodes".transferPnPLeft.jobInterface.hotPressLeftPICKJob4_A.loadingDone := "Unit1.Em5.ControlNodes".transferPnPLeft.jobInterface.hotPressLeftPICKJob4_A.workingDone;
END_REGION

REGION Network 32: Transfer P&P Left Job Interface Working Done [Side Tape → Hot Press Left][A]
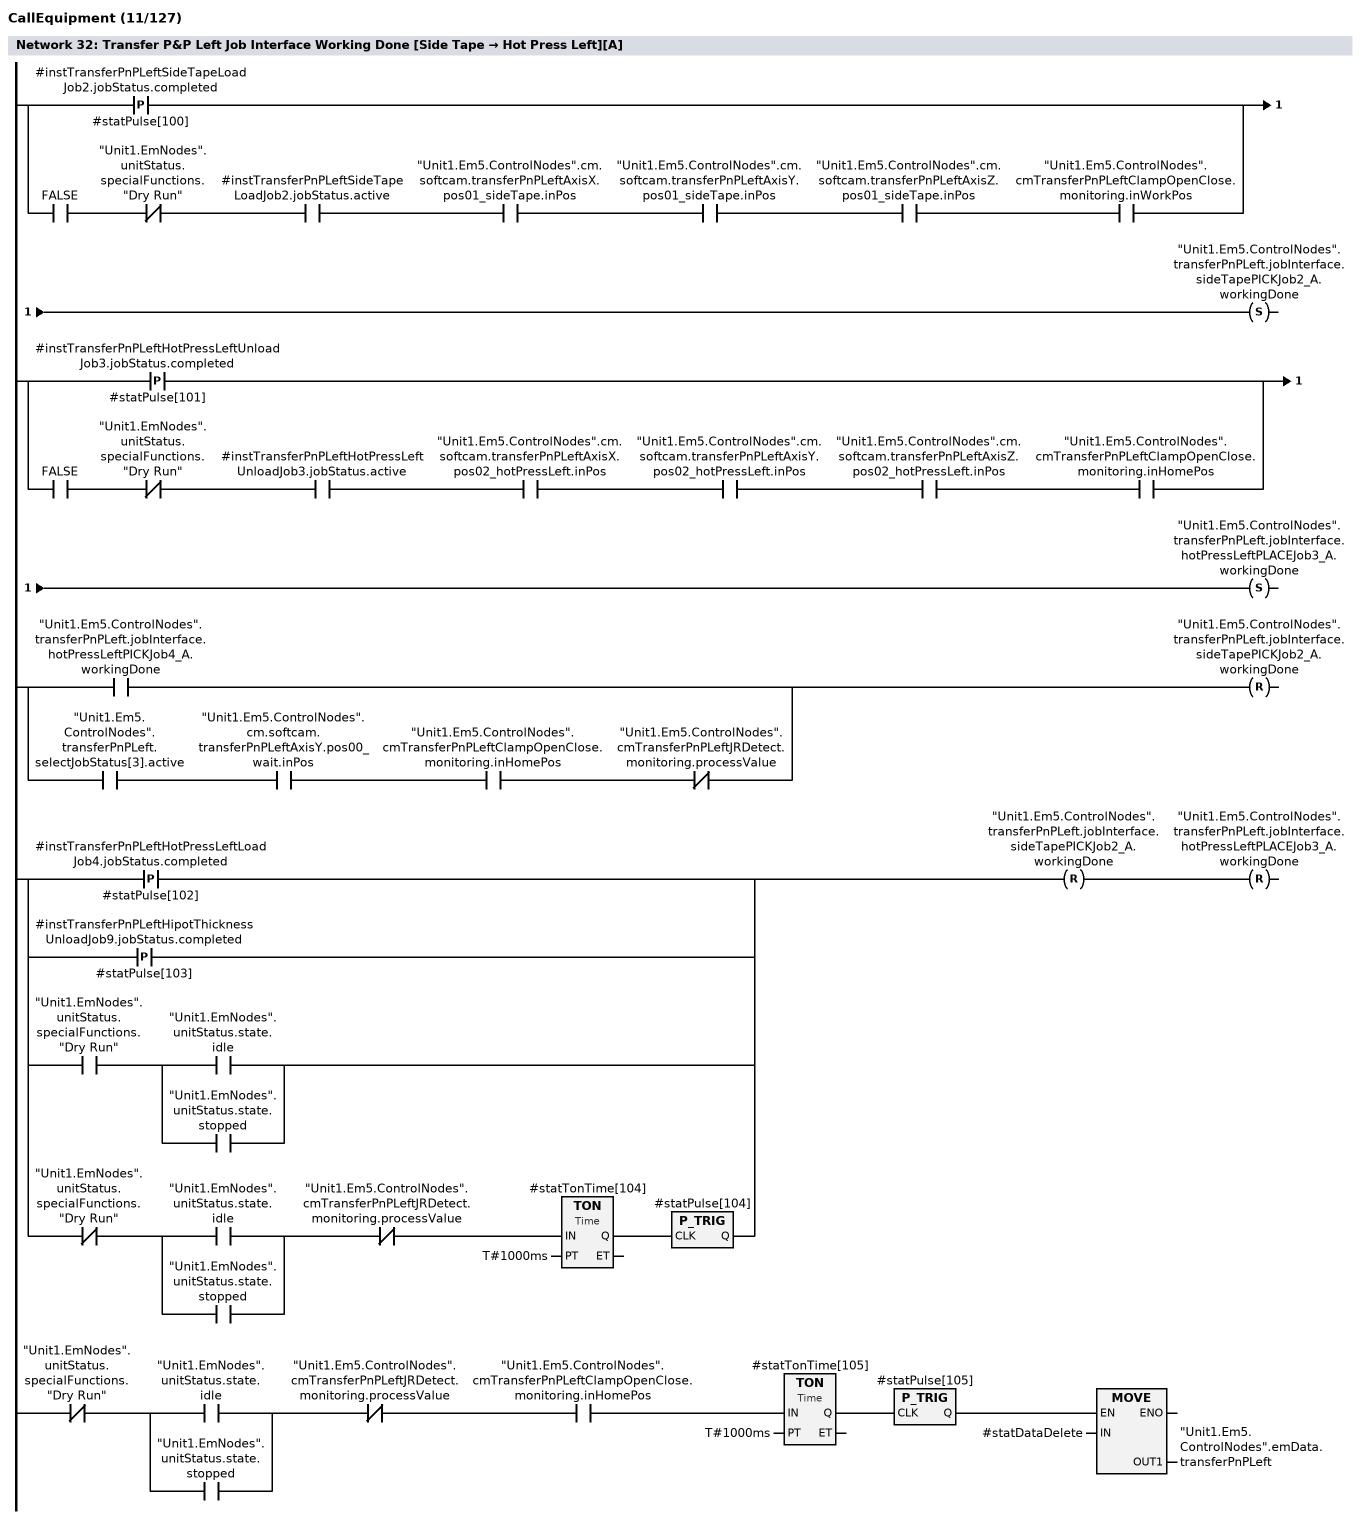
   RUNG wire#powerrail
      P_Contact(operand := #instTransferPnPLeftSideTapeLoadJob2.jobStatus.completed, bit := #statPulse[100])
      wire#w1
      S_Coil( "Unit1.Em5.ControlNodes".transferPnPLeft.jobInterface.sideTapePICKJob2_A.workingDone )
   END_RUNG
   RUNG wire#powerrail
      Contact( FALSE )
      I_Contact( "Unit1.EmNodes".unitStatus.specialFunctions."Dry Run" )
      Contact( #instTransferPnPLeftSideTapeLoadJob2.jobStatus.active )
      Contact( "Unit1.Em5.ControlNodes".cm.softcam.transferPnPLeftAxisX.pos01_sideTape.inPos )
      Contact( "Unit1.Em5.ControlNodes".cm.softcam.transferPnPLeftAxisY.pos01_sideTape.inPos )
      Contact( "Unit1.Em5.ControlNodes".cm.softcam.transferPnPLeftAxisZ.pos01_sideTape.inPos )
      Contact( "Unit1.Em5.ControlNodes".cmTransferPnPLeftClampOpenClose.monitoring.inWorkPos )
   END_RUNG wire#w1
   RUNG wire#powerrail
      P_Contact(operand := #instTransferPnPLeftHotPressLeftUnloadJob3.jobStatus.completed, bit := #statPulse[101])
      wire#w2
      S_Coil( "Unit1.Em5.ControlNodes".transferPnPLeft.jobInterface.hotPressLeftPLACEJob3_A.workingDone )
   END_RUNG
   RUNG wire#powerrail
      Contact( FALSE )
      I_Contact( "Unit1.EmNodes".unitStatus.specialFunctions."Dry Run" )
      Contact( #instTransferPnPLeftHotPressLeftUnloadJob3.jobStatus.active )
      Contact( "Unit1.Em5.ControlNodes".cm.softcam.transferPnPLeftAxisX.pos02_hotPressLeft.inPos )
      Contact( "Unit1.Em5.ControlNodes".cm.softcam.transferPnPLeftAxisY.pos02_hotPressLeft.inPos )
      Contact( "Unit1.Em5.ControlNodes".cm.softcam.transferPnPLeftAxisZ.pos02_hotPressLeft.inPos )
      Contact( "Unit1.Em5.ControlNodes".cmTransferPnPLeftClampOpenClose.monitoring.inHomePos )
   END_RUNG wire#w2
   RUNG wire#powerrail
      Contact( "Unit1.Em5.ControlNodes".transferPnPLeft.jobInterface.hotPressLeftPICKJob4_A.workingDone )
      wire#w3
      R_Coil( "Unit1.Em5.ControlNodes".transferPnPLeft.jobInterface.sideTapePICKJob2_A.workingDone )
   END_RUNG
   RUNG wire#powerrail
      Contact( "Unit1.Em5.ControlNodes".transferPnPLeft.selectJobStatus[3].active )
      Contact( "Unit1.Em5.ControlNodes".cm.softcam.transferPnPLeftAxisY.pos00_wait.inPos )
      Contact( "Unit1.Em5.ControlNodes".cmTransferPnPLeftClampOpenClose.monitoring.inHomePos )
      I_Contact( "Unit1.Em5.ControlNodes".cmTransferPnPLeftJRDetect.monitoring.processValue )
   END_RUNG wire#w3
   RUNG wire#powerrail
      P_Contact(operand := #instTransferPnPLeftHotPressLeftLoadJob4.jobStatus.completed, bit := #statPulse[102])
      wire#w4
      R_Coil( "Unit1.Em5.ControlNodes".transferPnPLeft.jobInterface.sideTapePICKJob2_A.workingDone )
      R_Coil( "Unit1.Em5.ControlNodes".transferPnPLeft.jobInterface.hotPressLeftPLACEJob3_A.workingDone )
   END_RUNG
   RUNG wire#powerrail
      P_Contact(operand := #instTransferPnPLeftHipotThicknessUnloadJob9.jobStatus.completed, bit := #statPulse[103])
   END_RUNG wire#w4
   RUNG wire#powerrail
      Contact( "Unit1.EmNodes".unitStatus.specialFunctions."Dry Run" )
      wire#w5
      Contact( "Unit1.EmNodes".unitStatus.state.idle )
   END_RUNG wire#w4
   RUNG wire#w5
      Contact( "Unit1.EmNodes".unitStatus.state.stopped )
   END_RUNG wire#w4
   RUNG wire#powerrail
      I_Contact( "Unit1.EmNodes".unitStatus.specialFunctions."Dry Run" )
      wire#w6
      Contact( "Unit1.EmNodes".unitStatus.state.idle )
      wire#w7
      I_Contact( "Unit1.Em5.ControlNodes".cmTransferPnPLeftJRDetect.monitoring.processValue )
      { S7_Templates := "time_type := Time" } #statTonTime[104].TON(pt := T#1000ms, et =>)
      P_Trig( #statPulse[104] )
   END_RUNG wire#w4
   RUNG wire#w6
      Contact( "Unit1.EmNodes".unitStatus.state.stopped )
   END_RUNG wire#w7
   RUNG wire#powerrail
      I_Contact( "Unit1.EmNodes".unitStatus.specialFunctions."Dry Run" )
      wire#w8
      Contact( "Unit1.EmNodes".unitStatus.state.idle )
      wire#w9
      I_Contact( "Unit1.Em5.ControlNodes".cmTransferPnPLeftJRDetect.monitoring.processValue )
      Contact( "Unit1.Em5.ControlNodes".cmTransferPnPLeftClampOpenClose.monitoring.inHomePos )
      { S7_Templates := "time_type := Time" } #statTonTime[105].TON(pt := T#1000ms, et =>)
      P_Trig( #statPulse[105] )
      Move(in := #statDataDelete, out1 => "Unit1.Em5.ControlNodes".emData.transferPnPLeft)
   END_RUNG
   RUNG wire#w8
      Contact( "Unit1.EmNodes".unitStatus.state.stopped )
   END_RUNG wire#w9
   // the same network as SCL:
   #_w1 := #instTransferPnPLeftSideTapeLoadJob2.jobStatus.completed AND NOT #statPulse[100];   // rising edge of #instTransferPnPLeftSideTapeLoadJob2.jobStatus.completed
   #statPulse[100] := #instTransferPnPLeftSideTapeLoadJob2.jobStatus.completed;
   IF #_w1 OR (FALSE AND NOT "Unit1.EmNodes".unitStatus.specialFunctions."Dry Run" AND #instTransferPnPLeftSideTapeLoadJob2.jobStatus.active AND "Unit1.Em5.ControlNodes".cm.softcam.transferPnPLeftAxisX.pos01_sideTape.inPos AND "Unit1.Em5.ControlNodes".cm.softcam.transferPnPLeftAxisY.pos01_sideTape.inPos AND "Unit1.Em5.ControlNodes".cm.softcam.transferPnPLeftAxisZ.pos01_sideTape.inPos AND "Unit1.Em5.ControlNodes".cmTransferPnPLeftClampOpenClose.monitoring.inWorkPos) THEN
       "Unit1.Em5.ControlNodes".transferPnPLeft.jobInterface.sideTapePICKJob2_A.workingDone := TRUE;
   END_IF;
   #_w2 := #instTransferPnPLeftHotPressLeftUnloadJob3.jobStatus.completed AND NOT #statPulse[101];   // rising edge of #instTransferPnPLeftHotPressLeftUnloadJob3.jobStatus.completed
   #statPulse[101] := #instTransferPnPLeftHotPressLeftUnloadJob3.jobStatus.completed;
   IF #_w2 OR (FALSE AND NOT "Unit1.EmNodes".unitStatus.specialFunctions."Dry Run" AND #instTransferPnPLeftHotPressLeftUnloadJob3.jobStatus.active AND "Unit1.Em5.ControlNodes".cm.softcam.transferPnPLeftAxisX.pos02_hotPressLeft.inPos AND "Unit1.Em5.ControlNodes".cm.softcam.transferPnPLeftAxisY.pos02_hotPressLeft.inPos AND "Unit1.Em5.ControlNodes".cm.softcam.transferPnPLeftAxisZ.pos02_hotPressLeft.inPos AND "Unit1.Em5.ControlNodes".cmTransferPnPLeftClampOpenClose.monitoring.inHomePos) THEN
       "Unit1.Em5.ControlNodes".transferPnPLeft.jobInterface.hotPressLeftPLACEJob3_A.workingDone := TRUE;
   END_IF;
   IF "Unit1.Em5.ControlNodes".transferPnPLeft.jobInterface.hotPressLeftPICKJob4_A.workingDone OR ("Unit1.Em5.ControlNodes".transferPnPLeft.selectJobStatus[3].active AND "Unit1.Em5.ControlNodes".cm.softcam.transferPnPLeftAxisY.pos00_wait.inPos AND "Unit1.Em5.ControlNodes".cmTransferPnPLeftClampOpenClose.monitoring.inHomePos AND NOT "Unit1.Em5.ControlNodes".cmTransferPnPLeftJRDetect.monitoring.processValue) THEN
       "Unit1.Em5.ControlNodes".transferPnPLeft.jobInterface.sideTapePICKJob2_A.workingDone := FALSE;
   END_IF;
   #_w3 := #instTransferPnPLeftHotPressLeftLoadJob4.jobStatus.completed AND NOT #statPulse[102];   // rising edge of #instTransferPnPLeftHotPressLeftLoadJob4.jobStatus.completed
   #statPulse[102] := #instTransferPnPLeftHotPressLeftLoadJob4.jobStatus.completed;
   #_w4 := #instTransferPnPLeftHipotThicknessUnloadJob9.jobStatus.completed AND NOT #statPulse[103];   // rising edge of #instTransferPnPLeftHipotThicknessUnloadJob9.jobStatus.completed
   #statPulse[103] := #instTransferPnPLeftHipotThicknessUnloadJob9.jobStatus.completed;
   #statTonTime[104].TON(IN := NOT "Unit1.EmNodes".unitStatus.specialFunctions."Dry Run" AND ("Unit1.EmNodes".unitStatus.state.idle OR "Unit1.EmNodes".unitStatus.state.stopped) AND NOT "Unit1.Em5.ControlNodes".cmTransferPnPLeftJRDetect.monitoring.processValue,
                         PT := T#1000ms);
   #_w5 := #statTonTime[104].Q AND NOT #statPulse[104];   // rising edge
   #statPulse[104] := #statTonTime[104].Q;
   IF #_w3 OR #_w4 OR ("Unit1.EmNodes".unitStatus.specialFunctions."Dry Run" AND ("Unit1.EmNodes".unitStatus.state.idle OR "Unit1.EmNodes".unitStatus.state.stopped)) OR #_w5 THEN
       "Unit1.Em5.ControlNodes".transferPnPLeft.jobInterface.sideTapePICKJob2_A.workingDone := FALSE;
       "Unit1.Em5.ControlNodes".transferPnPLeft.jobInterface.hotPressLeftPLACEJob3_A.workingDone := FALSE;
   END_IF;
   #statTonTime[105].TON(IN := NOT "Unit1.EmNodes".unitStatus.specialFunctions."Dry Run" AND ("Unit1.EmNodes".unitStatus.state.idle OR "Unit1.EmNodes".unitStatus.state.stopped) AND NOT "Unit1.Em5.ControlNodes".cmTransferPnPLeftJRDetect.monitoring.processValue AND "Unit1.Em5.ControlNodes".cmTransferPnPLeftClampOpenClose.monitoring.inHomePos,
                         PT := T#1000ms);
   #_w6 := #statTonTime[105].Q AND NOT #statPulse[105];   // rising edge
   #statPulse[105] := #statTonTime[105].Q;
   IF #_w6 THEN "Unit1.Em5.ControlNodes".emData.transferPnPLeft := #statDataDelete; END_IF;
END_REGION

REGION Network 34: [Job]Transfer P&P Left Select Job [BA40 - B]
   // Configure here when the jobs of the sequence should be started. More jobs could be added.
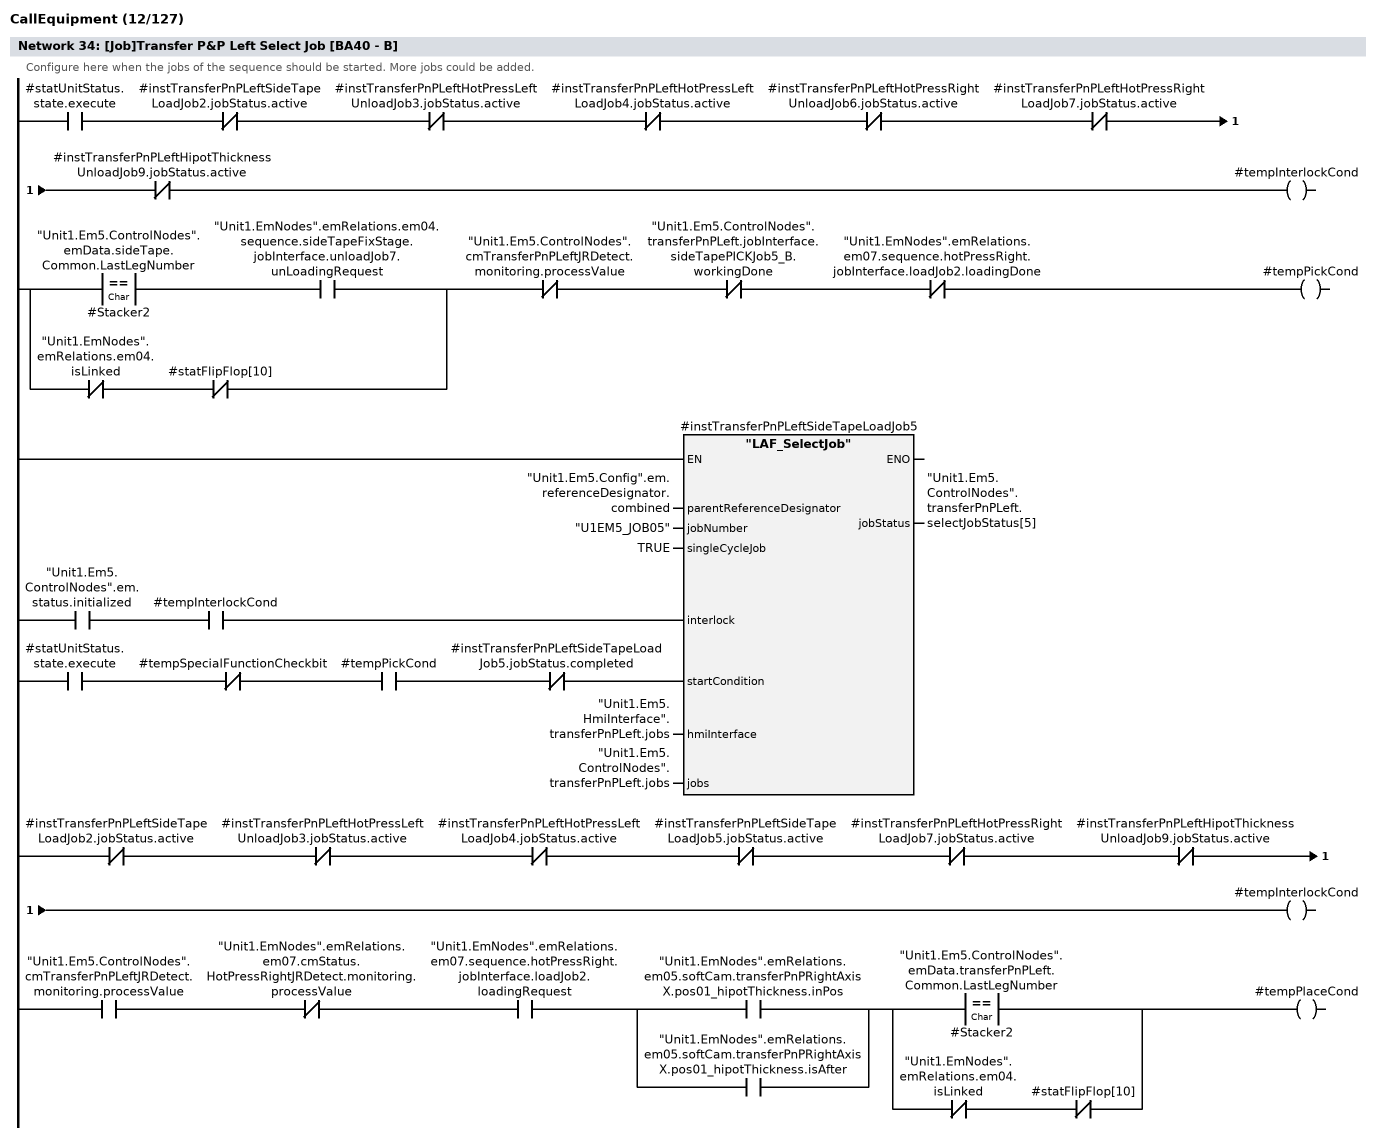
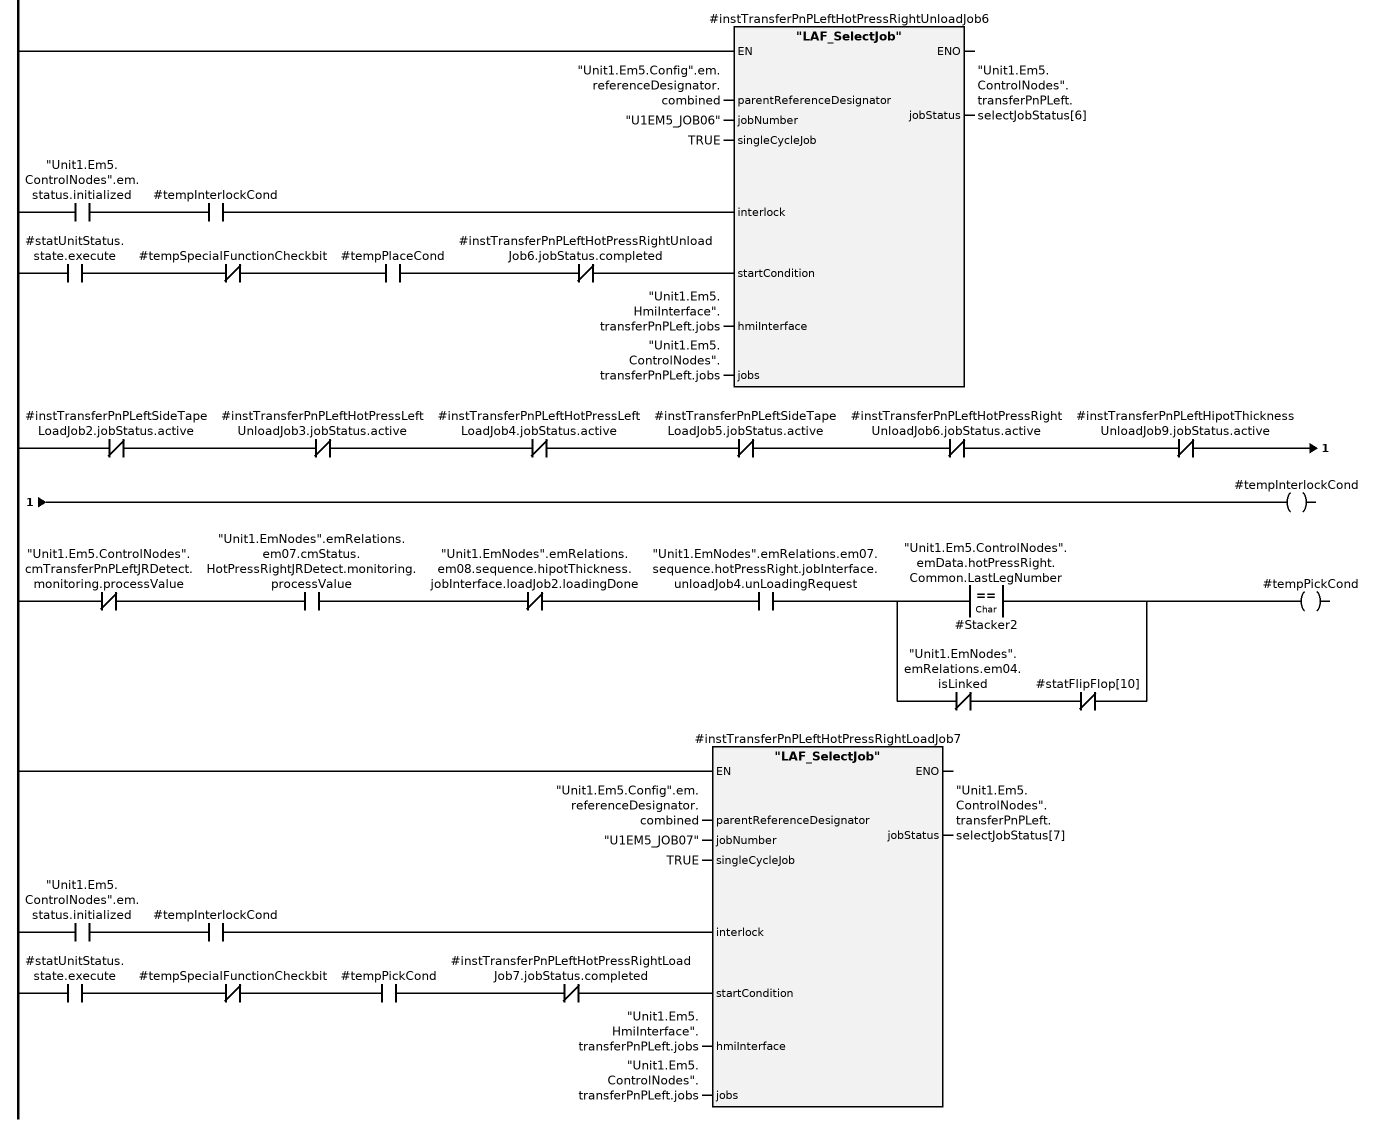
   RUNG wire#powerrail
      Contact( #statUnitStatus.state.execute )
      I_Contact( #instTransferPnPLeftSideTapeLoadJob2.jobStatus.active )
      I_Contact( #instTransferPnPLeftHotPressLeftUnloadJob3.jobStatus.active )
      I_Contact( #instTransferPnPLeftHotPressLeftLoadJob4.jobStatus.active )
      I_Contact( #instTransferPnPLeftHotPressRightUnloadJob6.jobStatus.active )
      I_Contact( #instTransferPnPLeftHotPressRightLoadJob7.jobStatus.active )
      I_Contact( #instTransferPnPLeftHipotThicknessUnloadJob9.jobStatus.active )
      Coil( #tempInterlockCond )
   END_RUNG
   RUNG wire#powerrail
      { S7_Templates := "SrcType := Char" } EQ_Contact(in1 := "Unit1.Em5.ControlNodes".emData.sideTape.Common.LastLegNumber, in2 := #Stacker2)
      Contact( "Unit1.EmNodes".emRelations.em04.sequence.sideTapeFixStage.jobInterface.unloadJob7.unLoadingRequest )
      wire#w1
      I_Contact( "Unit1.Em5.ControlNodes".cmTransferPnPLeftJRDetect.monitoring.processValue )
      I_Contact( "Unit1.Em5.ControlNodes".transferPnPLeft.jobInterface.sideTapePICKJob5_B.workingDone )
      I_Contact( "Unit1.EmNodes".emRelations.em07.sequence.hotPressRight.jobInterface.loadJob2.loadingDone )
      Coil( #tempPickCond )
   END_RUNG
   RUNG wire#powerrail
      I_Contact( "Unit1.EmNodes".emRelations.em04.isLinked )
      I_Contact( #statFlipFlop[10] )
   END_RUNG wire#w1
   RUNG wire#powerrail
      #instTransferPnPLeftSideTapeLoadJob5(interlock := wire#w2, startCondition := wire#w3, parentReferenceDesignator := "Unit1.Em5.Config".em.referenceDesignator.combined, jobNumber := "U1EM5_JOB05", singleCycleJob := TRUE, hmiInterface := "Unit1.Em5.HmiInterface".transferPnPLeft.jobs, jobs := "Unit1.Em5.ControlNodes".transferPnPLeft.jobs, jobStatus => "Unit1.Em5.ControlNodes".transferPnPLeft.selectJobStatus[5])
   END_RUNG
   RUNG wire#powerrail
      Contact( "Unit1.Em5.ControlNodes".em.status.initialized )
      Contact( #tempInterlockCond )
   END_RUNG wire#w2
   RUNG wire#powerrail
      Contact( #statUnitStatus.state.execute )
      I_Contact( #tempSpecialFunctionCheckbit )
      Contact( #tempPickCond )
      I_Contact( #instTransferPnPLeftSideTapeLoadJob5.jobStatus.completed )
   END_RUNG wire#w3
   RUNG wire#powerrail
      I_Contact( #instTransferPnPLeftSideTapeLoadJob2.jobStatus.active )
      I_Contact( #instTransferPnPLeftHotPressLeftUnloadJob3.jobStatus.active )
      I_Contact( #instTransferPnPLeftHotPressLeftLoadJob4.jobStatus.active )
      I_Contact( #instTransferPnPLeftSideTapeLoadJob5.jobStatus.active )
      I_Contact( #instTransferPnPLeftHotPressRightLoadJob7.jobStatus.active )
      I_Contact( #instTransferPnPLeftHipotThicknessUnloadJob9.jobStatus.active )
      Coil( #tempInterlockCond )
   END_RUNG
   RUNG wire#powerrail
      Contact( "Unit1.Em5.ControlNodes".cmTransferPnPLeftJRDetect.monitoring.processValue )
      I_Contact( "Unit1.EmNodes".emRelations.em07.cmStatus.HotPressRightJRDetect.monitoring.processValue )
      Contact( "Unit1.EmNodes".emRelations.em07.sequence.hotPressRight.jobInterface.loadJob2.loadingRequest )
      wire#w4
      Contact( "Unit1.EmNodes".emRelations.em05.softCam.transferPnPRightAxisX.pos01_hipotThickness.inPos )
      wire#w5
      { S7_Templates := "SrcType := Char" } EQ_Contact(in1 := "Unit1.Em5.ControlNodes".emData.transferPnPLeft.Common.LastLegNumber, in2 := #Stacker2)
      wire#w6
      Coil( #tempPlaceCond )
   END_RUNG
   RUNG wire#w4
      Contact( "Unit1.EmNodes".emRelations.em05.softCam.transferPnPRightAxisX.pos01_hipotThickness.isAfter )
   END_RUNG wire#w5
   RUNG wire#w5
      I_Contact( "Unit1.EmNodes".emRelations.em04.isLinked )
      I_Contact( #statFlipFlop[10] )
   END_RUNG wire#w6
   RUNG wire#powerrail
      #instTransferPnPLeftHotPressRightUnloadJob6(interlock := wire#w7, startCondition := wire#w8, parentReferenceDesignator := "Unit1.Em5.Config".em.referenceDesignator.combined, jobNumber := "U1EM5_JOB06", singleCycleJob := TRUE, hmiInterface := "Unit1.Em5.HmiInterface".transferPnPLeft.jobs, jobs := "Unit1.Em5.ControlNodes".transferPnPLeft.jobs, jobStatus => "Unit1.Em5.ControlNodes".transferPnPLeft.selectJobStatus[6])
   END_RUNG
   RUNG wire#powerrail
      Contact( "Unit1.Em5.ControlNodes".em.status.initialized )
      Contact( #tempInterlockCond )
   END_RUNG wire#w7
   RUNG wire#powerrail
      Contact( #statUnitStatus.state.execute )
      I_Contact( #tempSpecialFunctionCheckbit )
      Contact( #tempPlaceCond )
      I_Contact( #instTransferPnPLeftHotPressRightUnloadJob6.jobStatus.completed )
   END_RUNG wire#w8
   RUNG wire#powerrail
      I_Contact( #instTransferPnPLeftSideTapeLoadJob2.jobStatus.active )
      I_Contact( #instTransferPnPLeftHotPressLeftUnloadJob3.jobStatus.active )
      I_Contact( #instTransferPnPLeftHotPressLeftLoadJob4.jobStatus.active )
      I_Contact( #instTransferPnPLeftSideTapeLoadJob5.jobStatus.active )
      I_Contact( #instTransferPnPLeftHotPressRightUnloadJob6.jobStatus.active )
      I_Contact( #instTransferPnPLeftHipotThicknessUnloadJob9.jobStatus.active )
      Coil( #tempInterlockCond )
   END_RUNG
   RUNG wire#powerrail
      I_Contact( "Unit1.Em5.ControlNodes".cmTransferPnPLeftJRDetect.monitoring.processValue )
      Contact( "Unit1.EmNodes".emRelations.em07.cmStatus.HotPressRightJRDetect.monitoring.processValue )
      I_Contact( "Unit1.EmNodes".emRelations.em08.sequence.hipotThickness.jobInterface.loadJob2.loadingDone )
      Contact( "Unit1.EmNodes".emRelations.em07.sequence.hotPressRight.jobInterface.unloadJob4.unLoadingRequest )
      wire#w9
      { S7_Templates := "SrcType := Char" } EQ_Contact(in1 := "Unit1.Em5.ControlNodes".emData.hotPressRight.Common.LastLegNumber, in2 := #Stacker2)
      wire#w10
      Coil( #tempPickCond )
   END_RUNG
   RUNG wire#w9
      I_Contact( "Unit1.EmNodes".emRelations.em04.isLinked )
      I_Contact( #statFlipFlop[10] )
   END_RUNG wire#w10
   RUNG wire#powerrail
      #instTransferPnPLeftHotPressRightLoadJob7(interlock := wire#w11, startCondition := wire#w12, parentReferenceDesignator := "Unit1.Em5.Config".em.referenceDesignator.combined, jobNumber := "U1EM5_JOB07", singleCycleJob := TRUE, hmiInterface := "Unit1.Em5.HmiInterface".transferPnPLeft.jobs, jobs := "Unit1.Em5.ControlNodes".transferPnPLeft.jobs, jobStatus => "Unit1.Em5.ControlNodes".transferPnPLeft.selectJobStatus[7])
   END_RUNG
   RUNG wire#powerrail
      Contact( "Unit1.Em5.ControlNodes".em.status.initialized )
      Contact( #tempInterlockCond )
   END_RUNG wire#w11
   RUNG wire#powerrail
      Contact( #statUnitStatus.state.execute )
      I_Contact( #tempSpecialFunctionCheckbit )
      Contact( #tempPickCond )
      I_Contact( #instTransferPnPLeftHotPressRightLoadJob7.jobStatus.completed )
   END_RUNG wire#w12
   // the same network as SCL:
   #tempInterlockCond := #statUnitStatus.state.execute AND NOT #instTransferPnPLeftSideTapeLoadJob2.jobStatus.active AND NOT #instTransferPnPLeftHotPressLeftUnloadJob3.jobStatus.active AND NOT #instTransferPnPLeftHotPressLeftLoadJob4.jobStatus.active AND NOT #instTransferPnPLeftHotPressRightUnloadJob6.jobStatus.active AND NOT #instTransferPnPLeftHotPressRightLoadJob7.jobStatus.active AND NOT #instTransferPnPLeftHipotThicknessUnloadJob9.jobStatus.active;
   #tempPickCond := ((("Unit1.Em5.ControlNodes".emData.sideTape.Common.LastLegNumber = #Stacker2) AND "Unit1.EmNodes".emRelations.em04.sequence.sideTapeFixStage.jobInterface.unloadJob7.unLoadingRequest) OR (NOT "Unit1.EmNodes".emRelations.em04.isLinked AND NOT #statFlipFlop[10])) AND NOT "Unit1.Em5.ControlNodes".cmTransferPnPLeftJRDetect.monitoring.processValue AND NOT "Unit1.Em5.ControlNodes".transferPnPLeft.jobInterface.sideTapePICKJob5_B.workingDone AND NOT "Unit1.EmNodes".emRelations.em07.sequence.hotPressRight.jobInterface.loadJob2.loadingDone;
   #instTransferPnPLeftSideTapeLoadJob5(parentReferenceDesignator := "Unit1.Em5.Config".em.referenceDesignator.combined,   // "LAF_SelectJob"
                           jobNumber := "U1EM5_JOB05",
                           singleCycleJob := TRUE,
                           interlock := "Unit1.Em5.ControlNodes".em.status.initialized AND #tempInterlockCond,
                           startCondition := #statUnitStatus.state.execute AND NOT #tempSpecialFunctionCheckbit AND #tempPickCond AND NOT #instTransferPnPLeftSideTapeLoadJob5.jobStatus.completed,
                           hmiInterface := "Unit1.Em5.HmiInterface".transferPnPLeft.jobs,
                           jobs := "Unit1.Em5.ControlNodes".transferPnPLeft.jobs,
                           jobStatus => "Unit1.Em5.ControlNodes".transferPnPLeft.selectJobStatus[5]);
   #tempInterlockCond := NOT #instTransferPnPLeftSideTapeLoadJob2.jobStatus.active AND NOT #instTransferPnPLeftHotPressLeftUnloadJob3.jobStatus.active AND NOT #instTransferPnPLeftHotPressLeftLoadJob4.jobStatus.active AND NOT #instTransferPnPLeftSideTapeLoadJob5.jobStatus.active AND NOT #instTransferPnPLeftHotPressRightLoadJob7.jobStatus.active AND NOT #instTransferPnPLeftHipotThicknessUnloadJob9.jobStatus.active;
   #tempPlaceCond := "Unit1.Em5.ControlNodes".cmTransferPnPLeftJRDetect.monitoring.processValue AND NOT "Unit1.EmNodes".emRelations.em07.cmStatus.HotPressRightJRDetect.monitoring.processValue AND "Unit1.EmNodes".emRelations.em07.sequence.hotPressRight.jobInterface.loadJob2.loadingRequest AND ("Unit1.EmNodes".emRelations.em05.softCam.transferPnPRightAxisX.pos01_hipotThickness.inPos OR "Unit1.EmNodes".emRelations.em05.softCam.transferPnPRightAxisX.pos01_hipotThickness.isAfter) AND (("Unit1.Em5.ControlNodes".emData.transferPnPLeft.Common.LastLegNumber = #Stacker2) OR (NOT "Unit1.EmNodes".emRelations.em04.isLinked AND NOT #statFlipFlop[10]));
   #instTransferPnPLeftHotPressRightUnloadJob6(parentReferenceDesignator := "Unit1.Em5.Config".em.referenceDesignator.combined,   // "LAF_SelectJob"
                           jobNumber := "U1EM5_JOB06",
                           singleCycleJob := TRUE,
                           interlock := "Unit1.Em5.ControlNodes".em.status.initialized AND #tempInterlockCond,
                           startCondition := #statUnitStatus.state.execute AND NOT #tempSpecialFunctionCheckbit AND #tempPlaceCond AND NOT #instTransferPnPLeftHotPressRightUnloadJob6.jobStatus.completed,
                           hmiInterface := "Unit1.Em5.HmiInterface".transferPnPLeft.jobs,
                           jobs := "Unit1.Em5.ControlNodes".transferPnPLeft.jobs,
                           jobStatus => "Unit1.Em5.ControlNodes".transferPnPLeft.selectJobStatus[6]);
   #tempInterlockCond := NOT #instTransferPnPLeftSideTapeLoadJob2.jobStatus.active AND NOT #instTransferPnPLeftHotPressLeftUnloadJob3.jobStatus.active AND NOT #instTransferPnPLeftHotPressLeftLoadJob4.jobStatus.active AND NOT #instTransferPnPLeftSideTapeLoadJob5.jobStatus.active AND NOT #instTransferPnPLeftHotPressRightUnloadJob6.jobStatus.active AND NOT #instTransferPnPLeftHipotThicknessUnloadJob9.jobStatus.active;
   #tempPickCond := NOT "Unit1.Em5.ControlNodes".cmTransferPnPLeftJRDetect.monitoring.processValue AND "Unit1.EmNodes".emRelations.em07.cmStatus.HotPressRightJRDetect.monitoring.processValue AND NOT "Unit1.EmNodes".emRelations.em08.sequence.hipotThickness.jobInterface.loadJob2.loadingDone AND "Unit1.EmNodes".emRelations.em07.sequence.hotPressRight.jobInterface.unloadJob4.unLoadingRequest AND (("Unit1.Em5.ControlNodes".emData.hotPressRight.Common.LastLegNumber = #Stacker2) OR (NOT "Unit1.EmNodes".emRelations.em04.isLinked AND NOT #statFlipFlop[10]));
   #instTransferPnPLeftHotPressRightLoadJob7(parentReferenceDesignator := "Unit1.Em5.Config".em.referenceDesignator.combined,   // "LAF_SelectJob"
                           jobNumber := "U1EM5_JOB07",
                           singleCycleJob := TRUE,
                           interlock := "Unit1.Em5.ControlNodes".em.status.initialized AND #tempInterlockCond,
                           startCondition := #statUnitStatus.state.execute AND NOT #tempSpecialFunctionCheckbit AND #tempPickCond AND NOT #instTransferPnPLeftHotPressRightLoadJob7.jobStatus.completed,
                           hmiInterface := "Unit1.Em5.HmiInterface".transferPnPLeft.jobs,
                           jobs := "Unit1.Em5.ControlNodes".transferPnPLeft.jobs,
                           jobStatus => "Unit1.Em5.ControlNodes".transferPnPLeft.selectJobStatus[7]);
END_REGION

REGION Network 35: Transfer P&P Left Job Interface [Side Tape Loading][B]
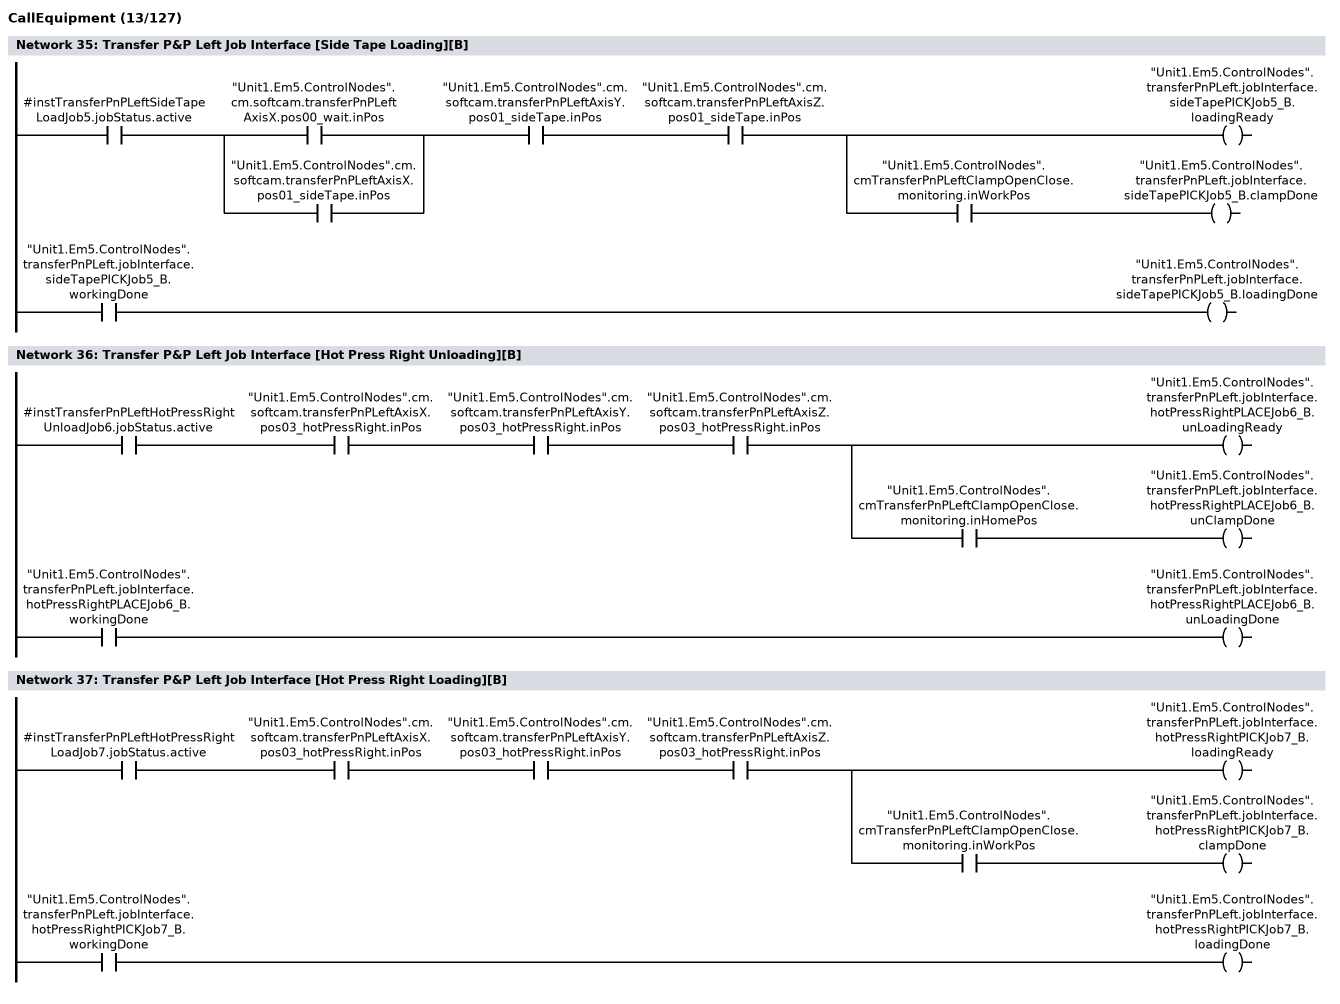
   RUNG wire#powerrail
      Contact( #instTransferPnPLeftSideTapeLoadJob5.jobStatus.active )
      wire#w1
      Contact( "Unit1.Em5.ControlNodes".cm.softcam.transferPnPLeftAxisX.pos00_wait.inPos )
      wire#w2
      Contact( "Unit1.Em5.ControlNodes".cm.softcam.transferPnPLeftAxisY.pos01_sideTape.inPos )
      Contact( "Unit1.Em5.ControlNodes".cm.softcam.transferPnPLeftAxisZ.pos01_sideTape.inPos )
      wire#w3
      Coil( "Unit1.Em5.ControlNodes".transferPnPLeft.jobInterface.sideTapePICKJob5_B.loadingReady )
   END_RUNG
   RUNG wire#w1
      Contact( "Unit1.Em5.ControlNodes".cm.softcam.transferPnPLeftAxisX.pos01_sideTape.inPos )
   END_RUNG wire#w2
   RUNG wire#w3
      Contact( "Unit1.Em5.ControlNodes".cmTransferPnPLeftClampOpenClose.monitoring.inWorkPos )
      Coil( "Unit1.Em5.ControlNodes".transferPnPLeft.jobInterface.sideTapePICKJob5_B.clampDone )
   END_RUNG
   RUNG wire#powerrail
      Contact( "Unit1.Em5.ControlNodes".transferPnPLeft.jobInterface.sideTapePICKJob5_B.workingDone )
      Coil( "Unit1.Em5.ControlNodes".transferPnPLeft.jobInterface.sideTapePICKJob5_B.loadingDone )
   END_RUNG
   // the same network as SCL:
   "Unit1.Em5.ControlNodes".transferPnPLeft.jobInterface.sideTapePICKJob5_B.loadingReady := #instTransferPnPLeftSideTapeLoadJob5.jobStatus.active AND ("Unit1.Em5.ControlNodes".cm.softcam.transferPnPLeftAxisX.pos00_wait.inPos OR "Unit1.Em5.ControlNodes".cm.softcam.transferPnPLeftAxisX.pos01_sideTape.inPos) AND "Unit1.Em5.ControlNodes".cm.softcam.transferPnPLeftAxisY.pos01_sideTape.inPos AND "Unit1.Em5.ControlNodes".cm.softcam.transferPnPLeftAxisZ.pos01_sideTape.inPos;
   "Unit1.Em5.ControlNodes".transferPnPLeft.jobInterface.sideTapePICKJob5_B.clampDone := "Unit1.Em5.ControlNodes".transferPnPLeft.jobInterface.sideTapePICKJob5_B.loadingReady AND "Unit1.Em5.ControlNodes".cmTransferPnPLeftClampOpenClose.monitoring.inWorkPos;
   "Unit1.Em5.ControlNodes".transferPnPLeft.jobInterface.sideTapePICKJob5_B.loadingDone := "Unit1.Em5.ControlNodes".transferPnPLeft.jobInterface.sideTapePICKJob5_B.workingDone;
END_REGION

REGION Network 36: Transfer P&P Left Job Interface [Hot Press Right Unloading][B]
   RUNG wire#powerrail
      Contact( #instTransferPnPLeftHotPressRightUnloadJob6.jobStatus.active )
      Contact( "Unit1.Em5.ControlNodes".cm.softcam.transferPnPLeftAxisX.pos03_hotPressRight.inPos )
      Contact( "Unit1.Em5.ControlNodes".cm.softcam.transferPnPLeftAxisY.pos03_hotPressRight.inPos )
      Contact( "Unit1.Em5.ControlNodes".cm.softcam.transferPnPLeftAxisZ.pos03_hotPressRight.inPos )
      wire#w1
      Coil( "Unit1.Em5.ControlNodes".transferPnPLeft.jobInterface.hotPressRightPLACEJob6_B.unLoadingReady )
   END_RUNG
   RUNG wire#w1
      Contact( "Unit1.Em5.ControlNodes".cmTransferPnPLeftClampOpenClose.monitoring.inHomePos )
      Coil( "Unit1.Em5.ControlNodes".transferPnPLeft.jobInterface.hotPressRightPLACEJob6_B.unClampDone )
   END_RUNG
   RUNG wire#powerrail
      Contact( "Unit1.Em5.ControlNodes".transferPnPLeft.jobInterface.hotPressRightPLACEJob6_B.workingDone )
      Coil( "Unit1.Em5.ControlNodes".transferPnPLeft.jobInterface.hotPressRightPLACEJob6_B.unLoadingDone )
   END_RUNG
   // the same network as SCL:
   "Unit1.Em5.ControlNodes".transferPnPLeft.jobInterface.hotPressRightPLACEJob6_B.unLoadingReady := #instTransferPnPLeftHotPressRightUnloadJob6.jobStatus.active AND "Unit1.Em5.ControlNodes".cm.softcam.transferPnPLeftAxisX.pos03_hotPressRight.inPos AND "Unit1.Em5.ControlNodes".cm.softcam.transferPnPLeftAxisY.pos03_hotPressRight.inPos AND "Unit1.Em5.ControlNodes".cm.softcam.transferPnPLeftAxisZ.pos03_hotPressRight.inPos;
   "Unit1.Em5.ControlNodes".transferPnPLeft.jobInterface.hotPressRightPLACEJob6_B.unClampDone := "Unit1.Em5.ControlNodes".transferPnPLeft.jobInterface.hotPressRightPLACEJob6_B.unLoadingReady AND "Unit1.Em5.ControlNodes".cmTransferPnPLeftClampOpenClose.monitoring.inHomePos;
   "Unit1.Em5.ControlNodes".transferPnPLeft.jobInterface.hotPressRightPLACEJob6_B.unLoadingDone := "Unit1.Em5.ControlNodes".transferPnPLeft.jobInterface.hotPressRightPLACEJob6_B.workingDone;
END_REGION

REGION Network 37: Transfer P&P Left Job Interface [Hot Press Right Loading][B]
   RUNG wire#powerrail
      Contact( #instTransferPnPLeftHotPressRightLoadJob7.jobStatus.active )
      Contact( "Unit1.Em5.ControlNodes".cm.softcam.transferPnPLeftAxisX.pos03_hotPressRight.inPos )
      Contact( "Unit1.Em5.ControlNodes".cm.softcam.transferPnPLeftAxisY.pos03_hotPressRight.inPos )
      Contact( "Unit1.Em5.ControlNodes".cm.softcam.transferPnPLeftAxisZ.pos03_hotPressRight.inPos )
      wire#w1
      Coil( "Unit1.Em5.ControlNodes".transferPnPLeft.jobInterface.hotPressRightPICKJob7_B.loadingReady )
   END_RUNG
   RUNG wire#w1
      Contact( "Unit1.Em5.ControlNodes".cmTransferPnPLeftClampOpenClose.monitoring.inWorkPos )
      Coil( "Unit1.Em5.ControlNodes".transferPnPLeft.jobInterface.hotPressRightPICKJob7_B.clampDone )
   END_RUNG
   RUNG wire#powerrail
      Contact( "Unit1.Em5.ControlNodes".transferPnPLeft.jobInterface.hotPressRightPICKJob7_B.workingDone )
      Coil( "Unit1.Em5.ControlNodes".transferPnPLeft.jobInterface.hotPressRightPICKJob7_B.loadingDone )
   END_RUNG
   // the same network as SCL:
   "Unit1.Em5.ControlNodes".transferPnPLeft.jobInterface.hotPressRightPICKJob7_B.loadingReady := #instTransferPnPLeftHotPressRightLoadJob7.jobStatus.active AND "Unit1.Em5.ControlNodes".cm.softcam.transferPnPLeftAxisX.pos03_hotPressRight.inPos AND "Unit1.Em5.ControlNodes".cm.softcam.transferPnPLeftAxisY.pos03_hotPressRight.inPos AND "Unit1.Em5.ControlNodes".cm.softcam.transferPnPLeftAxisZ.pos03_hotPressRight.inPos;
   "Unit1.Em5.ControlNodes".transferPnPLeft.jobInterface.hotPressRightPICKJob7_B.clampDone := "Unit1.Em5.ControlNodes".transferPnPLeft.jobInterface.hotPressRightPICKJob7_B.loadingReady AND "Unit1.Em5.ControlNodes".cmTransferPnPLeftClampOpenClose.monitoring.inWorkPos;
   "Unit1.Em5.ControlNodes".transferPnPLeft.jobInterface.hotPressRightPICKJob7_B.loadingDone := "Unit1.Em5.ControlNodes".transferPnPLeft.jobInterface.hotPressRightPICKJob7_B.workingDone;
END_REGION

REGION Network 38: Transfer P&P Left Job Interface Working Done [Side Tape → Hot Press Right][B]
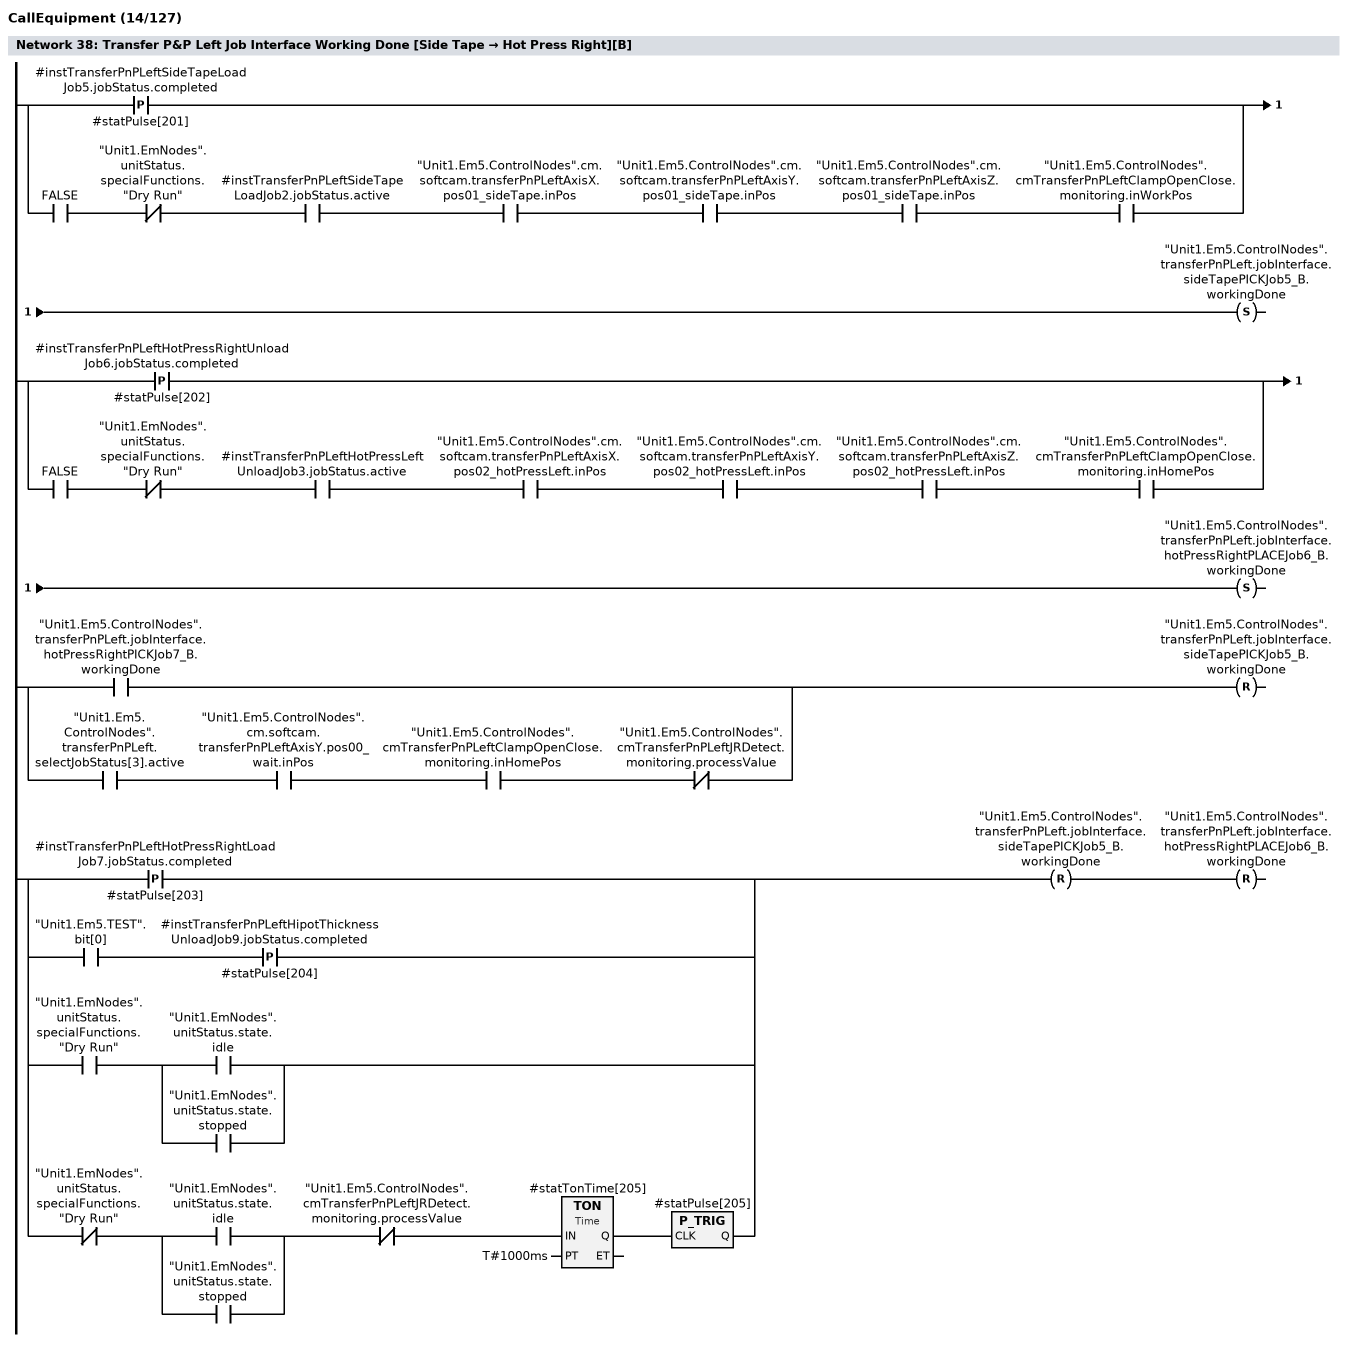
   RUNG wire#powerrail
      P_Contact(operand := #instTransferPnPLeftSideTapeLoadJob5.jobStatus.completed, bit := #statPulse[201])
      wire#w1
      S_Coil( "Unit1.Em5.ControlNodes".transferPnPLeft.jobInterface.sideTapePICKJob5_B.workingDone )
   END_RUNG
   RUNG wire#powerrail
      Contact( FALSE )
      I_Contact( "Unit1.EmNodes".unitStatus.specialFunctions."Dry Run" )
      Contact( #instTransferPnPLeftSideTapeLoadJob2.jobStatus.active )
      Contact( "Unit1.Em5.ControlNodes".cm.softcam.transferPnPLeftAxisX.pos01_sideTape.inPos )
      Contact( "Unit1.Em5.ControlNodes".cm.softcam.transferPnPLeftAxisY.pos01_sideTape.inPos )
      Contact( "Unit1.Em5.ControlNodes".cm.softcam.transferPnPLeftAxisZ.pos01_sideTape.inPos )
      Contact( "Unit1.Em5.ControlNodes".cmTransferPnPLeftClampOpenClose.monitoring.inWorkPos )
   END_RUNG wire#w1
   RUNG wire#powerrail
      P_Contact(operand := #instTransferPnPLeftHotPressRightUnloadJob6.jobStatus.completed, bit := #statPulse[202])
      wire#w2
      S_Coil( "Unit1.Em5.ControlNodes".transferPnPLeft.jobInterface.hotPressRightPLACEJob6_B.workingDone )
   END_RUNG
   RUNG wire#powerrail
      Contact( FALSE )
      I_Contact( "Unit1.EmNodes".unitStatus.specialFunctions."Dry Run" )
      Contact( #instTransferPnPLeftHotPressLeftUnloadJob3.jobStatus.active )
      Contact( "Unit1.Em5.ControlNodes".cm.softcam.transferPnPLeftAxisX.pos02_hotPressLeft.inPos )
      Contact( "Unit1.Em5.ControlNodes".cm.softcam.transferPnPLeftAxisY.pos02_hotPressLeft.inPos )
      Contact( "Unit1.Em5.ControlNodes".cm.softcam.transferPnPLeftAxisZ.pos02_hotPressLeft.inPos )
      Contact( "Unit1.Em5.ControlNodes".cmTransferPnPLeftClampOpenClose.monitoring.inHomePos )
   END_RUNG wire#w2
   RUNG wire#powerrail
      Contact( "Unit1.Em5.ControlNodes".transferPnPLeft.jobInterface.hotPressRightPICKJob7_B.workingDone )
      wire#w3
      R_Coil( "Unit1.Em5.ControlNodes".transferPnPLeft.jobInterface.sideTapePICKJob5_B.workingDone )
   END_RUNG
   RUNG wire#powerrail
      Contact( "Unit1.Em5.ControlNodes".transferPnPLeft.selectJobStatus[3].active )
      Contact( "Unit1.Em5.ControlNodes".cm.softcam.transferPnPLeftAxisY.pos00_wait.inPos )
      Contact( "Unit1.Em5.ControlNodes".cmTransferPnPLeftClampOpenClose.monitoring.inHomePos )
      I_Contact( "Unit1.Em5.ControlNodes".cmTransferPnPLeftJRDetect.monitoring.processValue )
   END_RUNG wire#w3
   RUNG wire#powerrail
      P_Contact(operand := #instTransferPnPLeftHotPressRightLoadJob7.jobStatus.completed, bit := #statPulse[203])
      wire#w4
      R_Coil( "Unit1.Em5.ControlNodes".transferPnPLeft.jobInterface.sideTapePICKJob5_B.workingDone )
      R_Coil( "Unit1.Em5.ControlNodes".transferPnPLeft.jobInterface.hotPressRightPLACEJob6_B.workingDone )
   END_RUNG
   RUNG wire#powerrail
      Contact( "Unit1.Em5.TEST".bit[0] )
      P_Contact(operand := #instTransferPnPLeftHipotThicknessUnloadJob9.jobStatus.completed, bit := #statPulse[204])
   END_RUNG wire#w4
   RUNG wire#powerrail
      Contact( "Unit1.EmNodes".unitStatus.specialFunctions."Dry Run" )
      wire#w5
      Contact( "Unit1.EmNodes".unitStatus.state.idle )
   END_RUNG wire#w4
   RUNG wire#w5
      Contact( "Unit1.EmNodes".unitStatus.state.stopped )
   END_RUNG wire#w4
   RUNG wire#powerrail
      I_Contact( "Unit1.EmNodes".unitStatus.specialFunctions."Dry Run" )
      wire#w6
      Contact( "Unit1.EmNodes".unitStatus.state.idle )
      wire#w7
      I_Contact( "Unit1.Em5.ControlNodes".cmTransferPnPLeftJRDetect.monitoring.processValue )
      { S7_Templates := "time_type := Time" } #statTonTime[205].TON(pt := T#1000ms, et =>)
      P_Trig( #statPulse[205] )
   END_RUNG wire#w4
   RUNG wire#w6
      Contact( "Unit1.EmNodes".unitStatus.state.stopped )
   END_RUNG wire#w7
   // the same network as SCL:
   #_w1 := #instTransferPnPLeftSideTapeLoadJob5.jobStatus.completed AND NOT #statPulse[201];   // rising edge of #instTransferPnPLeftSideTapeLoadJob5.jobStatus.completed
   #statPulse[201] := #instTransferPnPLeftSideTapeLoadJob5.jobStatus.completed;
   IF #_w1 OR (FALSE AND NOT "Unit1.EmNodes".unitStatus.specialFunctions."Dry Run" AND #instTransferPnPLeftSideTapeLoadJob2.jobStatus.active AND "Unit1.Em5.ControlNodes".cm.softcam.transferPnPLeftAxisX.pos01_sideTape.inPos AND "Unit1.Em5.ControlNodes".cm.softcam.transferPnPLeftAxisY.pos01_sideTape.inPos AND "Unit1.Em5.ControlNodes".cm.softcam.transferPnPLeftAxisZ.pos01_sideTape.inPos AND "Unit1.Em5.ControlNodes".cmTransferPnPLeftClampOpenClose.monitoring.inWorkPos) THEN
       "Unit1.Em5.ControlNodes".transferPnPLeft.jobInterface.sideTapePICKJob5_B.workingDone := TRUE;
   END_IF;
   #_w2 := #instTransferPnPLeftHotPressRightUnloadJob6.jobStatus.completed AND NOT #statPulse[202];   // rising edge of #instTransferPnPLeftHotPressRightUnloadJob6.jobStatus.completed
   #statPulse[202] := #instTransferPnPLeftHotPressRightUnloadJob6.jobStatus.completed;
   IF #_w2 OR (FALSE AND NOT "Unit1.EmNodes".unitStatus.specialFunctions."Dry Run" AND #instTransferPnPLeftHotPressLeftUnloadJob3.jobStatus.active AND "Unit1.Em5.ControlNodes".cm.softcam.transferPnPLeftAxisX.pos02_hotPressLeft.inPos AND "Unit1.Em5.ControlNodes".cm.softcam.transferPnPLeftAxisY.pos02_hotPressLeft.inPos AND "Unit1.Em5.ControlNodes".cm.softcam.transferPnPLeftAxisZ.pos02_hotPressLeft.inPos AND "Unit1.Em5.ControlNodes".cmTransferPnPLeftClampOpenClose.monitoring.inHomePos) THEN
       "Unit1.Em5.ControlNodes".transferPnPLeft.jobInterface.hotPressRightPLACEJob6_B.workingDone := TRUE;
   END_IF;
   IF "Unit1.Em5.ControlNodes".transferPnPLeft.jobInterface.hotPressRightPICKJob7_B.workingDone OR ("Unit1.Em5.ControlNodes".transferPnPLeft.selectJobStatus[3].active AND "Unit1.Em5.ControlNodes".cm.softcam.transferPnPLeftAxisY.pos00_wait.inPos AND "Unit1.Em5.ControlNodes".cmTransferPnPLeftClampOpenClose.monitoring.inHomePos AND NOT "Unit1.Em5.ControlNodes".cmTransferPnPLeftJRDetect.monitoring.processValue) THEN
       "Unit1.Em5.ControlNodes".transferPnPLeft.jobInterface.sideTapePICKJob5_B.workingDone := FALSE;
   END_IF;
   #_w3 := #instTransferPnPLeftHotPressRightLoadJob7.jobStatus.completed AND NOT #statPulse[203];   // rising edge of #instTransferPnPLeftHotPressRightLoadJob7.jobStatus.completed
   #statPulse[203] := #instTransferPnPLeftHotPressRightLoadJob7.jobStatus.completed;
   #_w4 := "Unit1.Em5.TEST".bit[0] AND #instTransferPnPLeftHipotThicknessUnloadJob9.jobStatus.completed AND NOT #statPulse[204];   // rising edge of #instTransferPnPLeftHipotThicknessUnloadJob9.jobStatus.completed
   #statPulse[204] := #instTransferPnPLeftHipotThicknessUnloadJob9.jobStatus.completed;
   #statTonTime[205].TON(IN := NOT "Unit1.EmNodes".unitStatus.specialFunctions."Dry Run" AND ("Unit1.EmNodes".unitStatus.state.idle OR "Unit1.EmNodes".unitStatus.state.stopped) AND NOT "Unit1.Em5.ControlNodes".cmTransferPnPLeftJRDetect.monitoring.processValue,
                         PT := T#1000ms);
   #_w5 := #statTonTime[205].Q AND NOT #statPulse[205];   // rising edge
   #statPulse[205] := #statTonTime[205].Q;
   IF #_w3 OR #_w4 OR ("Unit1.EmNodes".unitStatus.specialFunctions."Dry Run" AND ("Unit1.EmNodes".unitStatus.state.idle OR "Unit1.EmNodes".unitStatus.state.stopped)) OR #_w5 THEN
       "Unit1.Em5.ControlNodes".transferPnPLeft.jobInterface.sideTapePICKJob5_B.workingDone := FALSE;
       "Unit1.Em5.ControlNodes".transferPnPLeft.jobInterface.hotPressRightPLACEJob6_B.workingDone := FALSE;
   END_IF;
END_REGION

